KUKA KRL program: MyProgram_301().src

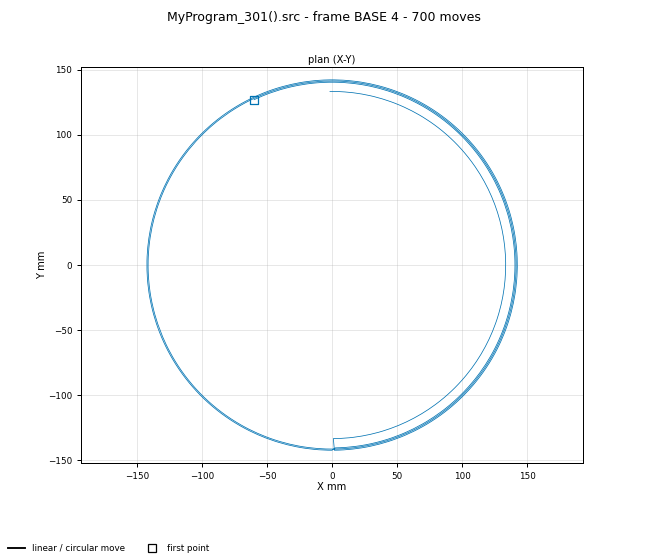
[picture p0: tool path of MyProgram_301().src in frame BASE 4, 700 of 700 moves have a stored position in this frame; points joined in program order, loops and branches not executed]
&ACCESS RVP
&REL 1
&PARAM TEMPLATE = C:\KRC\Roboter\Template\vorgabe
&PARAM EDITMASK = *
DEF MyProgram_301()
; ---- Setting reference (Base) ----
$BASE = BASE_DATA[4]

; --------------------------
; ---- Setting tool (TCP) ----
$TOOL = TOOL_DATA[3]
; --------------------------

$VEL.CP = VEL_APROX_PRINT
Startdeposition()
$VEL.CP = VEL_PRINT
LIN {X -59.9735,Y 127.061,Z 179,A 116.0898,B 5.4554,C 0.1242,E1 5.3915,E2 336.7382} C_DIS
LIN {X -56.1252,Y 128.8061,Z 179,A 114.464,B 5.4555,C 0.1213,E1 5.3956,E2 338.3506} C_DIS
LIN {X -53.7066,Y 129.8335,Z 179,A 112.9627,B 5.4555,C 0.1248,E1 5.3997,E2 339.9046} C_DIS
LIN {X -49.9072,Y 131.3417,Z 179,A 111.7575,B 5.4556,C 0.1181,E1 5.4027,E2 341.0513} C_DIS
LIN {X -46.6578,Y 132.5309,Z 179,A 110.2415,B 5.4556,C 0.1179,E1 5.4067,E2 342.5794} C_DIS
LIN {X -43.1664,Y 133.7078,Z 179,A 108.7239,B 5.4556,C 0.1168,E1 5.4107,E2 344.0979} C_DIS
LIN {X -39.9341,Y 134.7087,Z 179,A 107.5102,B 5.4557,C 0.1139,E1 5.4139,E2 345.2899} C_DIS
LIN {X -35.7865,Y 135.8693,Z 179,A 105.3832,B 5.4557,C 0.1168,E1 5.4197,E2 347.4621} C_DIS
LIN {X -31.4273,Y 136.9427,Z 179,A 103.8007,B 5.4557,C 0.1128,E1 5.4239,E2 349.0125} C_DIS
LIN {X -26.0499,Y 138.067,Z 179,A 101.4297,B 5.4557,C 0.1131,E1 5.4305,E2 351.3986} C_DIS
LIN {X -19.5272,Y 139.1395,Z 179,A 98.6974,B 5.4557,C 0.1125,E1 5.438,E2 354.1341} C_DIS
LIN {X -15.9211,Y 139.5996,Z 179,A 97.2765,B 5.4557,C 0.1113,E1 5.4419,E2 355.5466} C_DIS
LIN {X -11.8962,Y 139.9983,Z 179,A 95.031,B 5.4557,C 0.1179,E1 5.4484,E2 357.8653} C_DIS
LIN {X -6.6461,Y 140.3461,Z 179,A 93.5271,B 5.4557,C 0.1101,E1 5.4524,E2 359.2884} C_DIS
LIN {X -2.4559,Y 140.4815,Z 179,A 91.8062,B 5.4557,C 0.1102,E1 5.4572,E2 361.01} C_DIS
LIN {X 1.5144,Y 140.4967,Z 179,A 90.0682,B 5.4557,C 0.1117,E1 5.4621,E2 362.7621} C_DIS
LIN {X 5.4184,Y 140.3983,Z 179,A 88.5802,B 5.4557,C 0.1107,E1 5.4662,E2 364.2363} C_DIS
LIN {X 9.2875,Y 140.197,Z 179,A 86.9515,B 5.4557,C 0.1116,E1 5.4707,E2 365.8706} C_DIS
LIN {X 13.1744,Y 139.884,Z 179,A 85.4937,B 5.4557,C 0.1104,E1 5.4748,E2 367.3112} C_DIS
LIN {X 16.3822,Y 139.5446,Z 179,A 84.0811,B 5.4557,C 0.1121,E1 5.4787,E2 368.7355} C_DIS
LIN {X 22.469,Y 138.696,Z 179,A 81.6529,B 5.4557,C 0.1122,E1 5.4854,E2 371.1532} C_DIS
LIN {X 25.5598,Y 138.1606,Z 179,A 80.3615,B 5.4557,C 0.1131,E1 5.4889,E2 372.4458} C_DIS
LIN {X 29.0062,Y 137.4774,Z 179,A 78.85,B 5.4557,C 0.1149,E1 5.4931,E2 373.9666} C_DIS
LIN {X 36.0406,Y 135.8015,Z 179,A 75.9709,B 5.4557,C 0.1162,E1 5.5009,E2 376.8363} C_DIS
LIN {X 39.1776,Y 134.9302,Z 179,A 74.6743,B 5.4557,C 0.1169,E1 5.5044,E2 378.1288} C_DIS
LIN {X 42.5413,Y 133.9075,Z 179,A 73.2661,B 5.4557,C 0.1178,E1 5.5081,E2 379.5334} C_DIS
LIN {X 46.6696,Y 132.5268,Z 179,A 71.4197,B 5.4556,C 0.1204,E1 5.513,E2 381.3885} C_DIS
LIN {X 50.862,Y 130.9732,Z 179,A 69.7391,B 5.4556,C 0.1204,E1 5.5174,E2 383.0509} C_DIS
LIN {X 53.3945,Y 129.9638,Z 179,A 68.5414,B 5.4556,C 0.1228,E1 5.5205,E2 384.2594} C_DIS
LIN {X 57.312,Y 128.2819,Z 179,A 66.859,B 5.4555,C 0.1241,E1 5.5248,E2 385.9344} C_DIS
LIN {X 60.3668,Y 126.8731,Z 179,A 65.3438,B 5.4554,C 0.1277,E1 5.5287,E2 387.4675} C_DIS
LIN {X 65.3482,Y 124.3805,Z 179,A 63.2344,B 5.4554,C 0.1285,E1 5.5338,E2 389.5565} C_DIS
LIN {X 69.2323,Y 122.2642,Z 179,A 61.367,B 5.4553,C 0.1319,E1 5.5384,E2 391.432} C_DIS
LIN {X 73.1963,Y 119.9327,Z 179,A 59.5251,B 5.4553,C 0.1343,E1 5.5428,E2 393.2696} C_DIS
LIN {X 77.189,Y 117.4024,Z 179,A 57.7001,B 5.4553,C 0.1359,E1 5.5471,E2 395.0817} C_DIS
LIN {X 79.755,Y 115.6749,Z 179,A 56.1319,B 5.455,C 0.1422,E1 5.5508,E2 396.6886} C_DIS
LIN {X 82.8776,Y 113.4589,Z 179,A 54.84,B 5.455,C 0.1411,E1 5.5536,E2 397.9467} C_DIS
LIN {X 86.6009,Y 110.6427,Z 179,A 53.0145,B 5.455,C 0.1433,E1 5.5576,E2 399.7626} C_DIS
LIN {X 89.4387,Y 108.3616,Z 179,A 51.5047,B 5.455,C 0.1464,E1 5.5609,E2 401.2758} C_DIS
LIN {X 93.026,Y 105.2977,Z 179,A 49.9215,B 5.455,C 0.1452,E1 5.5642,E2 402.8161} C_DIS
LIN {X 96.3391,Y 102.2751,Z 179,A 47.5816,B 5.4547,C 0.156,E1 5.5691,E2 405.221} C_DIS
LIN {X 99.0644,Y 99.6378,Z 179,A 46.3542,B 5.4547,C 0.1546,E1 5.5715,E2 406.4084} C_DIS
LIN {X 102.2103,Y 96.4081,Z 179,A 44.5458,B 5.4547,C 0.1579,E1 5.575,E2 408.2135} C_DIS
LIN {X 105.3889,Y 92.923,Z 179,A 42.6665,B 5.4545,C 0.1614,E1 5.5785,E2 410.0877} C_DIS
LIN {X 108.7726,Y 88.9378,Z 179,A 40.4479,B 5.4543,C 0.1673,E1 5.5824,E2 412.318} C_DIS
LIN {X 111.8854,Y 84.99,Z 179,A 38.5181,B 5.4543,C 0.1702,E1 5.5857,E2 414.2331} C_DIS
LIN {X 114.5403,Y 81.3767,Z 179,A 36.8119,B 5.4542,C 0.1726,E1 5.5885,E2 415.9244} C_DIS
LIN {X 116.9616,Y 77.8554,Z 179,A 35.0581,B 5.454,C 0.1769,E1 5.5912,E2 417.6803} C_DIS
LIN {X 119.4477,Y 73.9851,Z 179,A 33.1916,B 5.4539,C 0.1813,E1 5.594,E2 419.5463} C_DIS
LIN {X 123.0392,Y 67.8445,Z 179,A 30.388,B 5.4537,C 0.187,E1 5.5979,E2 422.3387} C_DIS
LIN {X 125.0407,Y 64.0769,Z 179,A 28.7804,B 5.4537,C 0.1894,E1 5.6,E2 423.9302} C_DIS
LIN {X 126.7841,Y 60.5532,Z 179,A 27.2752,B 5.4535,C 0.1921,E1 5.6018,E2 425.4235} C_DIS
LIN {X 128.1026,Y 57.7127,Z 179,A 25.9599,B 5.4534,C 0.1959,E1 5.6033,E2 426.7445} C_DIS
LIN {X 129.3593,Y 54.842,Z 179,A 24.752,B 5.4533,C 0.1982,E1 5.6047,E2 427.9441} C_DIS
LIN {X 131.4521,Y 49.6125,Z 179,A 22.4725,B 5.4531,C 0.204,E1 5.607,E2 430.2225} C_DIS
LIN {X 132.5214,Y 46.685,Z 179,A 21.1591,B 5.4529,C 0.2081,E1 5.6082,E2 431.5422} C_DIS
LIN {X 133.8417,Y 42.7474,Z 179,A 19.6275,B 5.4529,C 0.2102,E1 5.6095,E2 433.0539} C_DIS
LIN {X 134.7772,Y 39.7003,Z 179,A 18.3035,B 5.4527,C 0.2141,E1 5.6106,E2 434.3818} C_DIS
LIN {X 135.6851,Y 36.4773,Z 179,A 16.9623,B 5.4526,C 0.2175,E1 5.6116,E2 435.7207} C_DIS
LIN {X 136.9654,Y 31.328,Z 179,A 15.0592,B 5.4525,C 0.2195,E1 5.6129,E2 437.5915} C_DIS
LIN {X 137.5627,Y 28.5976,Z 179,A 13.7924,B 5.4523,C 0.2246,E1 5.6136,E2 438.8755} C_DIS
LIN {X 138.2642,Y 24.9809,Z 179,A 12.2857,B 5.4521,C 0.2289,E1 5.6144,E2 440.3837} C_DIS
LIN {X 138.8135,Y 21.7222,Z 179,A 10.1318,B 5.4514,C 0.245,E1 5.6154,E2 442.6421} C_DIS
LIN {X 139.6771,Y 15.2107,Z 179,A 8.3722,B 5.4517,C 0.2385,E1 5.6159,E2 444.2856} C_DIS
LIN {X 140.0458,Y 11.3331,Z 179,A 6.7108,B 5.4514,C 0.2441,E1 5.6163,E2 445.9576} C_DIS
LIN {X 140.3011,Y 7.5426,Z 179,A 5.2604,B 5.4514,C 0.247,E1 5.6165,E2 447.3964} C_DIS
LIN {X 140.456,Y 3.6373,Z 179,A 3.6834,B 5.4511,C 0.2513,E1 5.6167,E2 448.9724} C_DIS
LIN {X 140.5034,Y -0.4635,Z 179,A 2.0429,B 5.4509,C 0.2556,E1 5.6167,E2 450.61} C_DIS
LIN {X 140.4368,Y -4.3279,Z 179,A 0.5019,B 5.4507,C 0.2595,E1 5.6166,E2 452.1476} C_DIS
LIN {X 140.2489,Y -8.4451,Z 179,A -1.064,B 5.4506,C 0.2625,E1 5.6164,E2 453.6999} C_DIS
LIN {X 139.9762,Y -12.1572,Z 179,A -2.5142,B 5.4504,C 0.2658,E1 5.616,E2 455.1425} C_DIS
LIN {X 139.5744,Y -16.133,Z 179,A -4.1622,B 5.4502,C 0.2707,E1 5.6155,E2 456.7942} C_DIS
LIN {X 139.1835,Y -19.2196,Z 179,A -5.448,B 5.45,C 0.2746,E1 5.6151,E2 458.0834} C_DIS
LIN {X 138.6268,Y -22.8834,Z 179,A -6.915,B 5.4498,C 0.2782,E1 5.6144,E2 459.5458} C_DIS
LIN {X 137.1833,Y -30.3685,Z 179,A -10.6169,B 5.4489,C 0.296,E1 5.6123,E2 463.3273} C_DIS
LIN {X 135.7517,Y -36.2274,Z 179,A -12.5921,B 5.4489,C 0.2954,E1 5.6109,E2 465.2418} C_DIS
LIN {X 134.7367,Y -39.8384,Z 179,A -13.9222,B 5.4489,C 0.2965,E1 5.6099,E2 466.5472} C_DIS
LIN {X 133.4221,Y -44.0409,Z 179,A -15.4975,B 5.4488,C 0.298,E1 5.6086,E2 468.0953} C_DIS
LIN {X 132.3787,Y -47.0869,Z 179,A -16.8262,B 5.4486,C 0.3018,E1 5.6073,E2 469.4272} C_DIS
LIN {X 131.1053,Y -50.5221,Z 179,A -18.223,B 5.4484,C 0.3044,E1 5.606,E2 470.8125} C_DIS
LIN {X 129.8345,Y -53.7041,Z 179,A -19.6741,B 5.4482,C 0.3089,E1 5.6044,E2 472.272} C_DIS
LIN {X 128.4058,Y -57.035,Z 179,A -21.053,B 5.448,C 0.3113,E1 5.6029,E2 473.6392} C_DIS
LIN {X 126.9294,Y -60.249,Z 179,A -22.4718,B 5.4478,C 0.3147,E1 5.6012,E2 475.0561} C_DIS
LIN {X 125.3758,Y -63.4187,Z 179,A -23.8583,B 5.4477,C 0.3176,E1 5.5995,E2 476.4369} C_DIS
LIN {X 123.5537,Y -66.9039,Z 179,A -25.5318,B 5.4474,C 0.3228,E1 5.5973,E2 478.1211} C_DIS
LIN {X 121.2798,Y -70.9418,Z 179,A -27.2877,B 5.4472,C 0.3255,E1 5.5949,E2 479.8611} C_DIS
LIN {X 117.8636,Y -76.4829,Z 179,A -29.9034,B 5.4468,C 0.3315,E1 5.591,E2 482.474} C_DIS
LIN {X 113.5484,Y -82.7547,Z 179,A -33.0276,B 5.4464,C 0.3392,E1 5.586,E2 485.6037} C_DIS
LIN {X 109.5829,Y -87.9384,Z 179,A -35.5981,B 5.4461,C 0.3439,E1 5.5816,E2 488.1645} C_DIS
LIN {X 106.9374,Y -91.1366,Z 179,A -37.2627,B 5.4459,C 0.3473,E1 5.5786,E2 489.827} C_DIS
LIN {X 104.9464,Y -93.4232,Z 179,A -38.4441,B 5.4457,C 0.3492,E1 5.5764,E2 491.0023} C_DIS
LIN {X 100.8459,Y -97.8345,Z 179,A -40.8197,B 5.4455,C 0.3533,E1 5.5719,E2 493.3694} C_DIS
LIN {X 97.8304,Y -100.8498,Z 179,A -42.5591,B 5.4452,C 0.3569,E1 5.5684,E2 495.1103} C_DIS
LIN {X 94.6187,Y -103.8693,Z 179,A -44.3238,B 5.445,C 0.36,E1 5.5648,E2 496.8723} C_DIS
LIN {X 90.594,Y -107.3979,Z 179,A -46.5101,B 5.4448,C 0.3643,E1 5.5602,E2 499.0609} C_DIS
LIN {X 87.1907,Y -110.1789,Z 179,A -48.2227,B 5.4446,C 0.3665,E1 5.5565,E2 500.7645} C_DIS
LIN {X 83.8356,Y -112.7522,Z 179,A -49.9475,B 5.4444,C 0.3696,E1 5.5527,E2 502.4908} C_DIS
LIN {X 77.9866,Y -116.874,Z 179,A -52.8046,B 5.4441,C 0.3737,E1 5.5461,E2 505.3422} C_DIS
LIN {X 72.6793,Y -120.2463,Z 179,A -55.5121,B 5.4437,C 0.3799,E1 5.5396,E2 508.0707} C_DIS
LIN {X 69.8696,Y -121.9007,Z 179,A -56.8094,B 5.4436,C 0.3814,E1 5.5365,E2 509.3649} C_DIS
LIN {X 65.3965,Y -124.3551,Z 179,A -58.5675,B 5.4436,C 0.3799,E1 5.5323,E2 511.0816} C_DIS
LIN {X 62.8045,Y -125.6861,Z 179,A -59.8854,B 5.4434,C 0.3834,E1 5.5289,E2 512.4178} C_DIS
LIN {X 59.2382,Y -127.4041,Z 179,A -61.3852,B 5.4434,C 0.3839,E1 5.5252,E2 513.9035} C_DIS
LIN {X 56.4868,Y -128.6498,Z 179,A -62.7339,B 5.4432,C 0.3871,E1 5.5217,E2 515.2688} C_DIS
LIN {X 52.7311,Y -130.2321,Z 179,A -64.274,B 5.4432,C 0.3874,E1 5.5178,E2 516.7938} C_DIS
LIN {X 49.4106,Y -131.5277,Z 179,A -65.7168,B 5.4431,C 0.3889,E1 5.514,E2 518.2363} C_DIS
LIN {X 46.2712,Y -132.6649,Z 179,A -66.9721,B 5.4431,C 0.3889,E1 5.5107,E2 519.4783} C_DIS
LIN {X 43.0135,Y -133.7567,Z 179,A -68.3877,B 5.4429,C 0.3905,E1 5.507,E2 520.8969} C_DIS
LIN {X 38.5766,Y -135.1051,Z 179,A -70.4033,B 5.4427,C 0.3939,E1 5.5015,E2 522.9304} C_DIS
LIN {X 34.6216,Y -136.1701,Z 179,A -72.4941,B 5.4422,C 0.401,E1 5.4957,E2 525.0779} C_DIS
LIN {X 29.928,Y -137.2784,Z 179,A -73.9126,B 5.4426,C 0.3951,E1 5.4921,E2 526.425} C_DIS
LIN {X 26.1079,Y -138.0559,Z 179,A -75.5015,B 5.4426,C 0.3962,E1 5.4877,E2 528.0148} C_DIS
LIN {X 22.1736,Y -138.7435,Z 179,A -77.5834,B 5.442,C 0.4031,E1 5.4818,E2 530.1578} C_DIS
LIN {X 17.83,Y -139.3675,Z 179,A -78.9522,B 5.4424,C 0.3985,E1 5.4781,E2 531.4719} C_DIS
LIN {X 13.6739,Y -139.836,Z 179,A -80.5373,B 5.4424,C 0.3976,E1 5.4738,E2 533.0418} C_DIS
LIN {X 10.8007,Y -140.0882,Z 179,A -81.8644,B 5.4423,C 0.4,E1 5.47,E2 534.3897} C_DIS
LIN {X 6.6782,Y -140.3445,Z 179,A -83.5282,B 5.4423,C 0.4002,E1 5.4654,E2 536.0516} C_DIS
LIN {X 2.5643,Y -140.4797,Z 179,A -85.0032,B 5.4424,C 0.3979,E1 5.4613,E2 537.5002} C_DIS
LIN {X 2.5643,Y -140.4797,Z 179,A -85.0032,B 5.4424,C 0.3979,E1 5.4613,E2 537.5002} C_DIS
Enddeposition()
LIN {X 0.9995,Y -141.4027,Z 179,A -85.5688,B 5.4422,C 0.4002,E1 5.4597,E2 538.089} C_DIS
Startdeposition()
$VEL.CP = VEL_PRINT
LIN {X 4.3079,Y -141.3411,Z 179,A -83.7777,B 5.4426,C 0.3941,E1 5.4648,E2 536.2364} C_DIS
LIN {X 8.0416,Y -141.1788,Z 179,A -82.3225,B 5.4426,C 0.3945,E1 5.4689,E2 534.7885} C_DIS
LIN {X 10.4771,Y -141.0176,Z 179,A -81.2424,B 5.4427,C 0.393,E1 5.4719,E2 533.6954} C_DIS
LIN {X 13.695,Y -140.7415,Z 179,A -79.9223,B 5.4427,C 0.3923,E1 5.4756,E2 532.3731} C_DIS
LIN {X 18.1055,Y -140.2424,Z 179,A -78.054,B 5.4429,C 0.3905,E1 5.4808,E2 530.4943} C_DIS
LIN {X 21.9939,Y -139.6855,Z 179,A -76.6375,B 5.4428,C 0.392,E1 5.4847,E2 529.1007} C_DIS
LIN {X 25.7892,Y -139.0366,Z 179,A -75.0635,B 5.4428,C 0.3909,E1 5.489,E2 527.524} C_DIS
LIN {X 28.3252,Y -138.54,Z 179,A -73.9262,B 5.443,C 0.3889,E1 5.4921,E2 526.3737} C_DIS
LIN {X 34.9333,Y -137.023,Z 179,A -71.2683,B 5.443,C 0.388,E1 5.4994,E2 523.7262} C_DIS
LIN {X 38.5958,Y -136.0377,Z 179,A -69.4507,B 5.4434,C 0.3828,E1 5.5043,E2 521.8694} C_DIS
LIN {X 41.7903,Y -135.0902,Z 179,A -68.4169,B 5.4432,C 0.3859,E1 5.507,E2 520.8777} C_DIS
LIN {X 45.0381,Y -134.0422,Z 179,A -66.9833,B 5.4434,C 0.3838,E1 5.5108,E2 519.4363} C_DIS
LIN {X 48.6768,Y -132.7657,Z 179,A -65.4951,B 5.4434,C 0.3831,E1 5.5147,E2 517.9571} C_DIS
LIN {X 51.5748,Y -131.6653,Z 179,A -64.2322,B 5.4435,C 0.3816,E1 5.518,E2 516.6923} C_DIS
LIN {X 55.4697,Y -130.0737,Z 179,A -62.6111,B 5.4435,C 0.3807,E1 5.5221,E2 515.0813} C_DIS
LIN {X 58.2837,Y -128.8368,Z 179,A -61.3322,B 5.4437,C 0.3787,E1 5.5254,E2 513.797} C_DIS
LIN {X 61.5935,Y -127.2882,Z 179,A -59.8657,B 5.4439,C 0.3769,E1 5.5291,E2 512.3313} C_DIS
LIN {X 64.4708,Y -125.8538,Z 179,A -58.5722,B 5.4439,C 0.3752,E1 5.5323,E2 511.038} C_DIS
LIN {X 67.6591,Y -124.1708,Z 179,A -56.614,B 5.4446,C 0.3659,E1 5.5373,E2 509.011} C_DIS
LIN {X 71.7411,Y -121.8579,Z 179,A -55.1964,B 5.4443,C 0.37,E1 5.5406,E2 507.6577} C_DIS
LIN {X 75.4899,Y -119.5717,Z 179,A -53.4446,B 5.4445,C 0.3676,E1 5.5447,E2 505.9083} C_DIS
LIN {X 79.2527,Y -117.1116,Z 179,A -51.5254,B 5.4448,C 0.3631,E1 5.5492,E2 503.9742} C_DIS
LIN {X 82.4628,Y -114.8741,Z 179,A -50.2247,B 5.4447,C 0.3646,E1 5.5521,E2 502.7109} C_DIS
LIN {X 85.389,Y -112.716,Z 179,A -48.6509,B 5.445,C 0.3604,E1 5.5557,E2 501.1222} C_DIS
LIN {X 88.4591,Y -110.3235,Z 179,A -47.0465,B 5.4452,C 0.3571,E1 5.5592,E2 499.5128} C_DIS
LIN {X 91.7741,Y -107.5811,Z 179,A -45.3391,B 5.4454,C 0.3543,E1 5.5628,E2 497.8088} C_DIS
LIN {X 95.2955,Y -104.475,Z 179,A -43.5116,B 5.4455,C 0.3517,E1 5.5666,E2 495.9898} C_DIS
LIN {X 98.3118,Y -101.6411,Z 179,A -41.8441,B 5.4457,C 0.3484,E1 5.57,E2 494.3221} C_DIS
LIN {X 101.5,Y -98.4575,Z 179,A -39.9945,B 5.446,C 0.3442,E1 5.5736,E2 492.4676} C_DIS
LIN {X 104.7884,Y -94.95,Z 179,A -38.1227,B 5.4462,C 0.3411,E1 5.5771,E2 490.6045} C_DIS
LIN {X 107.6795,Y -91.6583,Z 179,A -36.4504,B 5.4464,C 0.3388,E1 5.5802,E2 488.9445} C_DIS
LIN {X 110.2359,Y -88.5677,Z 179,A -34.7304,B 5.4467,C 0.3336,E1 5.5832,E2 487.2102} C_DIS
LIN {X 114.336,Y -83.2074,Z 179,A -32.4216,B 5.4467,C 0.3338,E1 5.587,E2 484.9564} C_DIS
LIN {X 117.0989,Y -79.2715,Z 179,A -30.2178,B 5.4472,C 0.3252,E1 5.5906,E2 482.7165} C_DIS
LIN {X 119.5465,Y -75.5298,Z 179,A -28.2286,B 5.4476,C 0.318,E1 5.5936,E2 480.7017} C_DIS
LIN {X 121.3857,Y -72.5372,Z 179,A -27.19,B 5.4475,C 0.3204,E1 5.595,E2 479.7137} C_DIS
LIN {X 123.3717,Y -69.1057,Z 179,A -25.5315,B 5.4477,C 0.3156,E1 5.5973,E2 478.0467} C_DIS
LIN {X 125.4173,Y -65.3168,Z 179,A -23.8624,B 5.4479,C 0.3123,E1 5.5995,E2 476.3861} C_DIS
LIN {X 126.9466,Y -62.2912,Z 179,A -22.5008,B 5.4481,C 0.3089,E1 5.6012,E2 475.025} C_DIS
LIN {X 128.5114,Y -58.9959,Z 179,A -21.0728,B 5.4483,C 0.3058,E1 5.6029,E2 473.6024} C_DIS
LIN {X 129.9129,Y -55.8417,Z 179,A -19.6603,B 5.4485,C 0.3019,E1 5.6045,E2 472.1868} C_DIS
LIN {X 131.3582,Y -52.3535,Z 179,A -18.2356,B 5.4486,C 0.2995,E1 5.606,E2 470.7748} C_DIS
LIN {X 132.4579,Y -49.5025,Z 179,A -16.9874,B 5.4488,C 0.296,E1 5.6072,E2 469.5241} C_DIS
LIN {X 133.8629,Y -45.5732,Z 179,A -15.381,B 5.449,C 0.2927,E1 5.6087,E2 467.9277} C_DIS
LIN {X 134.7945,Y -42.7332,Z 179,A -13.5688,B 5.4497,C 0.2799,E1 5.6103,E2 466.0335} C_DIS
LIN {X 136.3125,Y -37.6132,Z 179,A -12.1345,B 5.4494,C 0.2855,E1 5.6113,E2 464.6954} C_DIS
LIN {X 137.1844,Y -34.2974,Z 179,A -10.7171,B 5.4496,C 0.2812,E1 5.6123,E2 463.2731} C_DIS
LIN {X 138.048,Y -30.6439,Z 179,A -9.2203,B 5.4498,C 0.2773,E1 5.6132,E2 461.7783} C_DIS
LIN {X 138.9256,Y -26.3697,Z 179,A -7.5013,B 5.45,C 0.2731,E1 5.6141,E2 460.0642} C_DIS
LIN {X 139.5935,Y -22.5785,Z 179,A -5.8441,B 5.4503,C 0.2672,E1 5.6149,E2 458.3928} C_DIS
LIN {X 140.2021,Y -18.4129,Z 179,A -4.2597,B 5.4505,C 0.2643,E1 5.6155,E2 456.8231} C_DIS
LIN {X 140.6466,Y -14.6442,Z 179,A -2.862,B 5.4505,C 0.2621,E1 5.6159,E2 455.4428} C_DIS
LIN {X 140.9084,Y -11.8539,Z 179,A -1.7325,B 5.4507,C 0.259,E1 5.6162,E2 454.3132} C_DIS
LIN {X 141.1762,Y -8.0844,Z 179,A -0.2635,B 5.4509,C 0.2556,E1 5.6164,E2 452.8513} C_DIS
LIN {X 141.3108,Y -5.2017,Z 179,A 0.8759,B 5.451,C 0.2527,E1 5.6166,E2 451.7149} C_DIS
LIN {X 141.3956,Y -1.8135,Z 179,A 2.3343,B 5.4512,C 0.2475,E1 5.6166,E2 450.2441} C_DIS
LIN {X 141.3891,Y 2.2053,Z 179,A 3.8559,B 5.4514,C 0.2445,E1 5.6166,E2 448.7354} C_DIS
LIN {X 141.2762,Y 6.0877,Z 179,A 5.3231,B 5.4515,C 0.2417,E1 5.6165,E2 447.2812} C_DIS
LIN {X 141.092,Y 9.4502,Z 179,A 6.8304,B 5.4518,C 0.2356,E1 5.6162,E2 445.754} C_DIS
LIN {X 140.7421,Y 13.6884,Z 179,A 8.4336,B 5.4519,C 0.2326,E1 5.6158,E2 444.1654} C_DIS
LIN {X 140.0507,Y 19.5367,Z 179,A 10.5523,B 5.452,C 0.23,E1 5.6151,E2 442.0804} C_DIS
LIN {X 139.6935,Y 21.9426,Z 179,A 11.7579,B 5.4523,C 0.2238,E1 5.6146,E2 440.845} C_DIS
LIN {X 139.0271,Y 25.8385,Z 179,A 13.1623,B 5.4523,C 0.2224,E1 5.6139,E2 439.4656} C_DIS
LIN {X 138.0468,Y 30.6493,Z 179,A 15.1393,B 5.4525,C 0.2171,E1 5.6127,E2 437.489} C_DIS
LIN {X 137.4441,Y 33.238,Z 179,A 16.1352,B 5.4526,C 0.2153,E1 5.6121,E2 436.503} C_DIS
LIN {X 136.5242,Y 36.8366,Z 179,A 17.791,B 5.4529,C 0.2089,E1 5.6109,E2 434.8264} C_DIS
LIN {X 135.1491,Y 41.5978,Z 179,A 19.6956,B 5.453,C 0.205,E1 5.6094,E2 432.9342} C_DIS
LIN {X 133.9089,Y 45.4383,Z 179,A 21.2219,B 5.4531,C 0.2023,E1 5.6081,E2 431.4214} C_DIS
LIN {X 132.8684,Y 48.392,Z 179,A 22.4659,B 5.4532,C 0.1992,E1 5.6069,E2 430.1798} C_DIS
LIN {X 131.3335,Y 52.4149,Z 179,A 24.0987,B 5.4533,C 0.1963,E1 5.6053,E2 428.5608} C_DIS
LIN {X 129.9658,Y 55.7193,Z 179,A 25.7295,B 5.4536,C 0.1897,E1 5.6035,E2 426.9053} C_DIS
LIN {X 128.1395,Y 59.8002,Z 179,A 27.374,B 5.4536,C 0.1876,E1 5.6016,E2 425.2818} C_DIS
LIN {X 126.6554,Y 62.8816,Z 179,A 28.709,B 5.4537,C 0.1848,E1 5.5999,E2 423.9528} C_DIS
LIN {X 124.9198,Y 66.2642,Z 179,A 30.2338,B 5.4538,C 0.1812,E1 5.598,E2 422.4294} C_DIS
LIN {X 122.5344,Y 70.58,Z 179,A 31.9634,B 5.4538,C 0.1803,E1 5.5957,E2 420.734} C_DIS
LIN {X 121.1409,Y 72.9456,Z 179,A 33.3015,B 5.4541,C 0.1742,E1 5.5937,E2 419.366} C_DIS
LIN {X 118.9743,Y 76.4283,Z 179,A 34.8972,B 5.4541,C 0.1712,E1 5.5913,E2 417.7782} C_DIS
LIN {X 116.8132,Y 79.6928,Z 179,A 36.5251,B 5.4543,C 0.1668,E1 5.5888,E2 416.1443} C_DIS
LIN {X 114.1533,Y 83.4581,Z 179,A 38.3746,B 5.4544,C 0.1627,E1 5.5858,E2 414.2966} C_DIS
LIN {X 111.3389,Y 87.1769,Z 179,A 41.0152,B 5.4549,C 0.1473,E1 5.5811,E2 411.5569} C_DIS
LIN {X 106.9212,Y 92.5423,Z 179,A 42.6786,B 5.4546,C 0.1582,E1 5.5783,E2 410.0434} C_DIS
LIN {X 104.2774,Y 95.5113,Z 179,A 44.5475,B 5.4548,C 0.151,E1 5.5748,E2 408.1407} C_DIS
LIN {X 101.2022,Y 98.7642,Z 179,A 46.3398,B 5.4548,C 0.1476,E1 5.5713,E2 406.3508} C_DIS
LIN {X 92.8002,Y 106.6972,Z 179,A 50.5701,B 5.4549,C 0.145,E1 5.5628,E2 402.1783} C_DIS
LIN {X 90.2409,Y 108.8701,Z 179,A 52.0081,B 5.455,C 0.1414,E1 5.5597,E2 400.7302} C_DIS
LIN {X 87.7377,Y 110.8981,Z 179,A 53.57,B 5.4552,C 0.1354,E1 5.5562,E2 399.1351} C_DIS
LIN {X 84.0274,Y 113.735,Z 179,A 55.4478,B 5.4552,C 0.1323,E1 5.552,E2 397.259} C_DIS
LIN {X 80.1939,Y 116.4693,Z 179,A 57.2469,B 5.4552,C 0.1307,E1 5.5479,E2 395.4738} C_DIS
LIN {X 76.7917,Y 118.7402,Z 179,A 58.8582,B 5.4553,C 0.1287,E1 5.5442,E2 393.8683} C_DIS
LIN {X 73.4381,Y 120.8431,Z 179,A 60.4892,B 5.4553,C 0.1259,E1 5.5403,E2 392.2339} C_DIS
LIN {X 69.5643,Y 123.1139,Z 179,A 62.3138,B 5.4555,C 0.1232,E1 5.5359,E2 390.4085} C_DIS
LIN {X 63.6906,Y 126.251,Z 179,A 64.8495,B 5.4555,C 0.1218,E1 5.5297,E2 387.8938} C_DIS
LIN {X 60.3586,Y 127.8782,Z 179,A 66.3343,B 5.4555,C 0.1201,E1 5.5259,E2 386.4114} C_DIS
LIN {X 57.216,Y 129.3144,Z 179,A 67.8739,B 5.4556,C 0.1166,E1 5.522,E2 384.8541} C_DIS
LIN {X 53.6713,Y 130.8269,Z 179,A 69.2707,B 5.4556,C 0.117,E1 5.5184,E2 383.4787} C_DIS
LIN {X 50.8579,Y 131.944,Z 179,A 70.5007,B 5.4556,C 0.1157,E1 5.5152,E2 382.2483} C_DIS
LIN {X 47.5256,Y 133.1807,Z 179,A 72.1401,B 5.4557,C 0.1116,E1 5.5109,E2 380.5835} C_DIS
LIN {X 43.1876,Y 134.6494,Z 179,A 73.8845,B 5.4557,C 0.1113,E1 5.5063,E2 378.8538} C_DIS
LIN {X 38.9181,Y 135.9474,Z 179,A 75.5456,B 5.4557,C 0.1118,E1 5.5019,E2 377.2121} C_DIS
LIN {X 34.6025,Y 137.107,Z 179,A 77.4304,B 5.4557,C 0.1094,E1 5.4967,E2 375.318} C_DIS
LIN {X 30.5262,Y 138.0734,Z 179,A 78.9833,B 5.4557,C 0.1101,E1 5.4926,E2 373.7842} C_DIS
LIN {X 28.1021,Y 138.5854,Z 179,A 80.1016,B 5.4557,C 0.1081,E1 5.4895,E2 372.6514} C_DIS
LIN {X 24.3134,Y 139.3014,Z 179,A 81.5785,B 5.4557,C 0.1083,E1 5.4854,E2 371.186} C_DIS
LIN {X 19.7106,Y 140.0258,Z 179,A 83.4815,B 5.4557,C 0.1072,E1 5.4802,E2 369.2816} C_DIS
LIN {X 16.3303,Y 140.4606,Z 179,A 84.7817,B 5.4557,C 0.1077,E1 5.4766,E2 367.9923} C_DIS
LIN {X 13.2086,Y 140.7882,Z 179,A 86.2109,B 5.4558,C 0.1053,E1 5.4726,E2 366.5434} C_DIS
LIN {X 8.9197,Y 141.1247,Z 179,A 87.9047,B 5.4558,C 0.1055,E1 5.4679,E2 364.8566} C_DIS
LIN {X 5.0338,Y 141.3174,Z 179,A 89.5584,B 5.4558,C 0.1043,E1 5.4632,E2 363.1937} C_DIS
LIN {X 0.5177,Y 141.4055,Z 179,A 91.3077,B 5.4558,C 0.1052,E1 5.4584,E2 361.4555} C_DIS
LIN {X -3.1022,Y 141.3742,Z 179,A 92.6987,B 5.4558,C 0.1061,E1 5.4545,E2 360.0749} C_DIS
LIN {X -6.3182,Y 141.2671,Z 179,A 94.2803,B 5.4558,C 0.1029,E1 5.45,E2 358.4584} C_DIS
LIN {X -10.6336,Y 141.0061,Z 179,A 95.7763,B 5.4558,C 0.1062,E1 5.4459,E2 356.996} C_DIS
LIN {X -14.818,Y 140.6279,Z 179,A 97.4476,B 5.4558,C 0.107,E1 5.4413,E2 355.3295} C_DIS
LIN {X -17.7046,Y 140.2949,Z 179,A 98.7868,B 5.4558,C 0.1054,E1 5.4375,E2 353.9702} C_DIS
LIN {X -22.2365,Y 139.6475,Z 179,A 101.0043,B 5.4558,C 0.1019,E1 5.4313,E2 351.7073} C_DIS
LIN {X -26.4875,Y 138.903,Z 179,A 102.3477,B 5.4558,C 0.1075,E1 5.4277,E2 350.4168} C_DIS
LIN {X -30.1852,Y 138.147,Z 179,A 103.8422,B 5.4558,C 0.1087,E1 5.4237,E2 348.9277} C_DIS
LIN {X -34.2779,Y 137.1893,Z 179,A 106.1026,B 5.4558,C 0.1034,E1 5.4174,E2 346.5968} C_DIS
LIN {X -39.0294,Y 135.9148,Z 179,A 107.4949,B 5.4558,C 0.1118,E1 5.4138,E2 345.283} C_DIS
LIN {X -42.3801,Y 134.9073,Z 179,A 108.9044,B 5.4557,C 0.113,E1 5.4101,E2 343.8754} C_DIS
LIN {X -45.1784,Y 133.9954,Z 179,A 110.173,B 5.4557,C 0.1132,E1 5.4067,E2 342.5978} C_DIS
LIN {X -49.121,Y 132.6008,Z 179,A 112.0412,B 5.4557,C 0.1128,E1 5.4017,E2 340.7086} C_DIS
LIN {X -52.9605,Y 131.1136,Z 179,A 113.6582,B 5.4557,C 0.1151,E1 5.3975,E2 339.0993} C_DIS
LIN {X -56.4558,Y 129.6474,Z 179,A 115.1341,B 5.4556,C 0.1174,E1 5.3938,E2 337.6321} C_DIS
LIN {X -59.8038,Y 128.1379,Z 179,A 116.6459,B 5.4556,C 0.1189,E1 5.3899,E2 336.1184} C_DIS
LIN {X -63.3872,Y 126.4055,Z 179,A 118.255,B 5.4556,C 0.1209,E1 5.3859,E2 334.5109} C_DIS
LIN {X -67.0537,Y 124.4988,Z 179,A 120.0426,B 5.4555,C 0.1219,E1 5.3814,E2 332.7101} C_DIS
LIN {X -71.0188,Y 122.2804,Z 179,A 121.9262,B 5.4555,C 0.124,E1 5.3769,E2 330.8224} C_DIS
LIN {X -75.0441,Y 119.8527,Z 179,A 123.8601,B 5.4554,C 0.1265,E1 5.3723,E2 328.8862} C_DIS
LIN {X -78.9175,Y 117.3385,Z 179,A 125.7741,B 5.4554,C 0.1289,E1 5.3678,E2 326.9682} C_DIS
LIN {X -85.6625,Y 112.5084,Z 179,A 128.8659,B 5.4551,C 0.1373,E1 5.3609,E2 323.9138} C_DIS
LIN {X -87.9222,Y 110.7513,Z 179,A 130.2927,B 5.4551,C 0.1365,E1 5.3577,E2 322.4538} C_DIS
LIN {X -91.1943,Y 108.0735,Z 179,A 132.4097,B 5.4551,C 0.1355,E1 5.353,E2 320.2863} C_DIS
LIN {X -94.2464,Y 105.4217,Z 179,A 133.904,B 5.4551,C 0.1401,E1 5.35,E2 318.8119} C_DIS
LIN {X -98.227,Y 101.7232,Z 179,A 136.0031,B 5.4549,C 0.1454,E1 5.3457,E2 316.7278} C_DIS
LIN {X -101.5761,Y 98.379,Z 179,A 138.2849,B 5.4549,C 0.1456,E1 5.3412,E2 314.4008} C_DIS
LIN {X -104.4166,Y 95.359,Z 179,A 139.7378,B 5.4548,C 0.1514,E1 5.3385,E2 312.9786} C_DIS
LIN {X -110.3474,Y 88.4294,Z 179,A 144.2085,B 5.4548,C 0.1518,E1 5.3304,E2 308.4106} C_DIS
LIN {X -114.2965,Y 83.2619,Z 179,A 145.8305,B 5.4543,C 0.1677,E1 5.3279,E2 306.9223} C_DIS
LIN {X -117.2668,Y 79.0235,Z 179,A 148.1978,B 5.4543,C 0.17,E1 5.3241,E2 304.5221} C_DIS
LIN {X -119.6034,Y 75.4398,Z 179,A 150.051,B 5.4541,C 0.173,E1 5.3213,E2 302.6549} C_DIS
LIN {X -122.0106,Y 71.4813,Z 179,A 151.9552,B 5.454,C 0.1774,E1 5.3185,E2 300.7489} C_DIS
LIN {X -124.3232,Y 67.3797,Z 179,A 154.1234,B 5.4539,C 0.1796,E1 5.3156,E2 298.5487} C_DIS
LIN {X -125.8307,Y 64.5163,Z 179,A 155.4705,B 5.4538,C 0.1826,E1 5.3139,E2 297.198} C_DIS
LIN {X -127.3722,Y 61.4177,Z 179,A 156.4633,B 5.4535,C 0.1901,E1 5.3127,E2 296.2594} C_DIS
LIN {X -129.2797,Y 57.2935,Z 179,A 158.5152,B 5.4535,C 0.1929,E1 5.3103,E2 294.1819} C_DIS
LIN {X -131.5415,Y 51.8933,Z 179,A 160.8546,B 5.4532,C 0.1995,E1 5.3078,E2 291.849} C_DIS
LIN {X -132.5521,Y 49.2509,Z 179,A 162.1209,B 5.4532,C 0.2014,E1 5.3066,E2 290.568} C_DIS
LIN {X -133.6876,Y 46.0789,Z 179,A 163.4986,B 5.453,C 0.2049,E1 5.3053,E2 289.1899} C_DIS
LIN {X -134.7082,Y 43.0035,Z 179,A 164.8781,B 5.4529,C 0.2079,E1 5.3041,E2 287.8028} C_DIS
LIN {X -135.9946,Y 38.7499,Z 179,A 166.6216,B 5.4527,C 0.2133,E1 5.3027,E2 286.0684} C_DIS
LIN {X -136.7897,Y 35.8407,Z 179,A 167.9215,B 5.4526,C 0.216,E1 5.3018,E2 284.7594} C_DIS
LIN {X -137.5055,Y 32.9831,Z 179,A 169.1618,B 5.4525,C 0.2189,E1 5.301,E2 283.5141} C_DIS
LIN {X -138.295,Y 29.4999,Z 179,A 171.3606,B 5.4525,C 0.2159,E1 5.2996,E2 281.2181} C_DIS
LIN {X -139.3643,Y 23.9522,Z 179,A 172.936,B 5.4521,C 0.229,E1 5.2989,E2 279.7382} C_DIS
LIN {X -139.7776,Y 21.3995,Z 179,A 174.1256,B 5.452,C 0.2306,E1 5.2984,E2 278.531} C_DIS
LIN {X -140.3853,Y 16.9614,Z 179,A 176.3124,B 5.452,C 0.2323,E1 5.2976,E2 276.297} C_DIS
LIN {X -140.7863,Y 13.2281,Z 179,A 177.5696,B 5.4516,C 0.2391,E1 5.2973,E2 275.0756} C_DIS
LIN {X -141.0724,Y 9.7259,Z 179,A 178.9252,B 5.4514,C 0.2437,E1 5.297,E2 273.73} C_DIS
LIN {X -141.2632,Y 6.3954,Z 179,A -179.6842,B 5.4513,C 0.2472,E1 5.2968,E2 272.3355} C_DIS
LIN {X -141.3607,Y 3.6021,Z 179,A -178.4224,B 5.4512,C 0.2493,E1 5.2967,E2 271.0576} C_DIS
LIN {X -141.3989,Y -1.5802,Z 179,A -176.0952,B 5.451,C 0.2531,E1 5.2967,E2 268.7022} C_DIS
LIN {X -141.2996,Y -5.4889,Z 179,A -174.635,B 5.4507,C 0.2588,E1 5.2968,E2 267.2595} C_DIS
LIN {X -141.0719,Y -9.7334,Z 179,A -172.7693,B 5.4506,C 0.2623,E1 5.2972,E2 265.3762} C_DIS
LIN {X -140.4728,Y -16.2277,Z 179,A -170.1651,B 5.4502,C 0.2702,E1 5.2979,E2 262.779} C_DIS
LIN {X -139.8416,Y -20.9861,Z 179,A -168.096,B 5.45,C 0.2745,E1 5.2987,E2 260.6949} C_DIS
LIN {X -139.3131,Y -24.248,Z 179,A -166.5884,B 5.4498,C 0.2766,E1 5.2994,E2 259.166} C_DIS
LIN {X -138.436,Y -28.8366,Z 179,A -164.9004,B 5.4495,C 0.2838,E1 5.3003,E2 257.5062} C_DIS
LIN {X -137.7649,Y -31.8844,Z 179,A -163.6107,B 5.4493,C 0.2871,E1 5.3011,E2 256.214} C_DIS
LIN {X -137.0373,Y -34.8771,Z 179,A -162.3238,B 5.4491,C 0.2901,E1 5.302,E2 254.9228} C_DIS
LIN {X -136.1721,Y -38.1152,Z 179,A -160.8821,B 5.449,C 0.293,E1 5.3031,E2 253.4708} C_DIS
LIN {X -134.9073,Y -42.3801,Z 179,A -159.143,B 5.4487,C 0.2985,E1 5.3045,E2 251.7413} C_DIS
LIN {X -133.9887,Y -45.1988,Z 179,A -157.8305,B 5.4486,C 0.3007,E1 5.3056,E2 250.4148} C_DIS
LIN {X -131.0661,Y -53.0783,Z 179,A -154.7493,B 5.4479,C 0.3128,E1 5.3086,E2 247.3784} C_DIS
LIN {X -130.2875,Y -54.9635,Z 179,A -153.4872,B 5.448,C 0.3108,E1 5.31,E2 246.0592} C_DIS
LIN {X -128.4471,Y -59.135,Z 179,A -151.8434,B 5.4476,C 0.3175,E1 5.3119,E2 244.4434} C_DIS
LIN {X -127.4658,Y -61.2217,Z 179,A -150.6354,B 5.4476,C 0.3172,E1 5.3134,E2 243.1996} C_DIS
LIN {X -125.6976,Y -64.7778,Z 179,A -148.9922,B 5.4474,C 0.3209,E1 5.3154,E2 241.5527} C_DIS
LIN {X -122.7235,Y -70.2504,Z 179,A -146.456,B 5.4471,C 0.327,E1 5.3189,E2 239.0161} C_DIS
LIN {X -120.7719,Y -73.5559,Z 179,A -144.7303,B 5.4469,C 0.329,E1 5.3214,E2 237.2683} C_DIS
LIN {X -118.3289,Y -77.4245,Z 179,A -142.8303,B 5.4467,C 0.3329,E1 5.3243,E2 235.363} C_DIS
LIN {X -115.767,Y -81.2051,Z 179,A -141.0106,B 5.4464,C 0.3374,E1 5.3271,E2 233.548} C_DIS
LIN {X -113.1811,Y -84.7722,Z 179,A -139.1586,B 5.4462,C 0.3407,E1 5.3302,E2 231.6877} C_DIS
LIN {X -110.6783,Y -88.0138,Z 179,A -137.4354,B 5.446,C 0.3437,E1 5.3332,E2 229.9565} C_DIS
LIN {X -107.754,Y -91.5707,Z 179,A -135.5278,B 5.4458,C 0.3472,E1 5.3366,E2 228.0438} C_DIS
LIN {X -104.8282,Y -94.9062,Z 179,A -133.6848,B 5.4456,C 0.3504,E1 5.3401,E2 226.1953} C_DIS
LIN {X -101.6507,Y -98.3019,Z 179,A -131.767,B 5.4454,C 0.3539,E1 5.3438,E2 224.2734} C_DIS
LIN {X -98.272,Y -101.6796,Z 179,A -129.8116,B 5.4452,C 0.3574,E1 5.3477,E2 222.3158} C_DIS
LIN {X -94.9086,Y -104.8261,Z 179,A -127.9305,B 5.4449,C 0.3607,E1 5.3515,E2 220.433} C_DIS
LIN {X -91.6647,Y -107.6741,Z 179,A -126.156,B 5.4448,C 0.3635,E1 5.3553,E2 218.6554} C_DIS
LIN {X -88.4076,Y -110.3649,Z 179,A -124.3717,B 5.4446,C 0.3656,E1 5.3592,E2 216.8616} C_DIS
LIN {X -84.3361,Y -113.5058,Z 179,A -122.4295,B 5.4443,C 0.3706,E1 5.3635,E2 214.9386} C_DIS
LIN {X -81.2673,Y -115.7231,Z 179,A -120.7232,B 5.4443,C 0.3711,E1 5.3674,E2 213.2092} C_DIS
LIN {X -77.4426,Y -118.317,Z 179,A -118.8712,B 5.444,C 0.3741,E1 5.3717,E2 211.3601} C_DIS
LIN {X -73.7782,Y -120.6356,Z 179,A -117.0476,B 5.444,C 0.3758,E1 5.376,E2 209.5275} C_DIS
LIN {X -69.8871,Y -122.9307,Z 179,A -114.9801,B 5.444,C 0.3756,E1 5.3811,E2 207.428} C_DIS
LIN {X -66.9346,Y -124.5628,Z 179,A -113.973,B 5.4435,C 0.3814,E1 5.3835,E2 206.4695} C_DIS
LIN {X -63.8442,Y -126.1728,Z 179,A -112.448,B 5.4435,C 0.3818,E1 5.3873,E2 204.929} C_DIS
LIN {X -60.3054,Y -127.9036,Z 179,A -110.8447,B 5.4434,C 0.3835,E1 5.3913,E2 203.3247} C_DIS
LIN {X -57.4714,Y -129.2002,Z 179,A -109.568,B 5.4434,C 0.3847,E1 5.3946,E2 202.0458} C_DIS
LIN {X -53.9333,Y -130.7178,Z 179,A -108.0188,B 5.4432,C 0.3863,E1 5.3986,E2 200.498} C_DIS
LIN {X -51.0028,Y -131.8876,Z 179,A -106.365,B 5.4434,C 0.3831,E1 5.403,E2 198.7931} C_DIS
LIN {X -47.5098,Y -133.1864,Z 179,A -104.878,B 5.4434,C 0.3846,E1 5.4069,E2 197.309} C_DIS
LIN {X -44.2066,Y -134.3191,Z 179,A -103.7565,B 5.443,C 0.3892,E1 5.4098,E2 196.227} C_DIS
LIN {X -39.8549,Y -135.6731,Z 179,A -101.7584,B 5.443,C 0.3887,E1 5.4152,E2 194.208} C_DIS
LIN {X -35.7977,Y -136.8012,Z 179,A -100.2132,B 5.4428,C 0.3917,E1 5.4193,E2 192.6842} C_DIS
LIN {X -32.749,Y -137.5619,Z 179,A -98.9596,B 5.4428,C 0.3927,E1 5.4227,E2 191.4328} C_DIS
LIN {X -29.1283,Y -138.3752,Z 179,A -97.4128,B 5.4428,C 0.3929,E1 5.4269,E2 189.8799} C_DIS
LIN {X -26.1918,Y -138.9596,Z 179,A -96.1374,B 5.4428,C 0.3926,E1 5.4305,E2 188.5956} C_DIS
LIN {X -22.407,Y -139.6216,Z 179,A -94.4774,B 5.4428,C 0.3919,E1 5.4351,E2 186.9211} C_DIS
LIN {X -18.1191,Y -140.2406,Z 179,A -92.7699,B 5.4428,C 0.3929,E1 5.4398,E2 185.2194} C_DIS
LIN {X -14.305,Y -140.6829,Z 179,A -91.3122,B 5.4426,C 0.3944,E1 5.4438,E2 183.7744} C_DIS
LIN {X -11.3424,Y -140.9516,Z 179,A -90.1291,B 5.4426,C 0.3949,E1 5.4471,E2 182.5939} C_DIS
LIN {X -8.3956,Y -141.157,Z 179,A -88.8326,B 5.4426,C 0.3937,E1 5.4507,E2 181.2834} C_DIS
LIN {X -4.8486,Y -141.3246,Z 179,A -87.4885,B 5.4426,C 0.3949,E1 5.4545,E2 179.9515} C_DIS
LIN {X -1.6214,Y -141.3988,Z 179,A -86.1865,B 5.4426,C 0.3949,E1 5.4581,E2 178.6497} C_DIS
LIN {X 0.9995,Y -141.4027,Z 179,A -85.5666,B 5.4422,C 0.4004,E1 5.4597,E2 178.0889} C_DIS
Enddeposition()
LIN {X 0.9995,Y -141.4027,Z 179,A -85.5666,B 5.4422,C 0.4004,E1 5.4597,E2 178.0889} C_DIS
Startdeposition()
$VEL.CP = VEL_PRINT
LIN {X 0.0013,Y -142.3117,Z 179,A -86.0551,B 5.442,C 0.4047,E1 5.4583,E2 178.622} C_DIS
LIN {X -3.2536,Y -142.2741,Z 179,A -87.3393,B 5.442,C 0.4044,E1 5.4547,E2 179.9032} C_DIS
LIN {X -6.9714,Y -142.1387,Z 179,A -88.849,B 5.442,C 0.4046,E1 5.4505,E2 181.4151} C_DIS
LIN {X -10.2874,Y -141.9372,Z 179,A -90.2616,B 5.4419,C 0.4055,E1 5.4465,E2 182.8385} C_DIS
LIN {X -13.715,Y -141.647,Z 179,A -91.6439,B 5.4419,C 0.4052,E1 5.4426,E2 184.2209} C_DIS
LIN {X -17.4145,Y -141.241,Z 179,A -93.096,B 5.4419,C 0.4044,E1 5.4386,E2 185.6674} C_DIS
LIN {X -20.6408,Y -140.8054,Z 179,A -94.4405,B 5.4419,C 0.4044,E1 5.4349,E2 187.0169} C_DIS
LIN {X -24.0878,Y -140.2575,Z 179,A -95.8892,B 5.4419,C 0.4044,E1 5.4309,E2 188.472} C_DIS
LIN {X -27.5336,Y -139.6227,Z 179,A -97.2643,B 5.442,C 0.4035,E1 5.4271,E2 189.8427} C_DIS
LIN {X -31.1724,Y -138.8542,Z 179,A -98.6955,B 5.4422,C 0.4019,E1 5.4232,E2 191.2654} C_DIS
LIN {X -34.3405,Y -138.1054,Z 179,A -100.0865,B 5.4422,C 0.4022,E1 5.4194,E2 192.6676} C_DIS
LIN {X -37.7142,Y -137.2222,Z 179,A -101.497,B 5.4422,C 0.4014,E1 5.4156,E2 194.0793} C_DIS
LIN {X -41.0661,Y -136.2565,Z 179,A -102.8131,B 5.4423,C 0.3994,E1 5.4121,E2 195.3838} C_DIS
LIN {X -44.0813,Y -135.3122,Z 179,A -104.2002,B 5.4423,C 0.3998,E1 5.4084,E2 196.7868} C_DIS
LIN {X -47.664,Y -134.0911,Z 179,A -105.6807,B 5.4424,C 0.3981,E1 5.4045,E2 198.2617} C_DIS
LIN {X -50.8466,Y -132.9176,Z 179,A -107.2088,B 5.4424,C 0.3988,E1 5.4005,E2 199.8119} C_DIS
LIN {X -54.4526,Y -131.4798,Z 179,A -108.6762,B 5.4426,C 0.3961,E1 5.3967,E2 201.2666} C_DIS
LIN {X -57.0544,Y -130.3727,Z 179,A -109.8209,B 5.4426,C 0.395,E1 5.3938,E2 202.4123} C_DIS
LIN {X -60.055,Y -129.0169,Z 179,A -111.1397,B 5.4428,C 0.3935,E1 5.3904,E2 203.7303} C_DIS
LIN {X -63.1952,Y -127.5079,Z 179,A -112.6022,B 5.4428,C 0.3926,E1 5.3867,E2 205.201} C_DIS
LIN {X -66.9099,Y -125.601,Z 179,A -114.288,B 5.443,C 0.3906,E1 5.3825,E2 206.8876} C_DIS
LIN {X -70.5746,Y -123.5785,Z 179,A -116.067,B 5.443,C 0.3895,E1 5.3782,E2 208.6792} C_DIS
LIN {X -74.5508,Y -121.2213,Z 179,A -117.913,B 5.4433,C 0.3868,E1 5.3738,E2 210.5231} C_DIS
LIN {X -78.2396,Y -118.8738,Z 179,A -119.6812,B 5.4434,C 0.3843,E1 5.3696,E2 212.2924} C_DIS
LIN {X -81.8416,Y -116.4234,Z 179,A -121.4617,B 5.4436,C 0.382,E1 5.3655,E2 214.0763} C_DIS
LIN {X -85.3689,Y -113.8629,Z 179,A -123.2727,B 5.4437,C 0.3798,E1 5.3614,E2 215.8948} C_DIS
LIN {X -88.8311,Y -111.1824,Z 179,A -125.0325,B 5.444,C 0.3768,E1 5.3575,E2 217.6539} C_DIS
LIN {X -91.7131,Y -108.8173,Z 179,A -126.6603,B 5.444,C 0.3755,E1 5.354,E2 219.2985} C_DIS
LIN {X -95.0559,Y -105.9094,Z 179,A -128.4538,B 5.4443,C 0.3724,E1 5.3503,E2 221.093} C_DIS
LIN {X -98.2198,Y -102.982,Z 179,A -130.2233,B 5.4444,C 0.3695,E1 5.3466,E2 222.8667} C_DIS
LIN {X -101.3286,Y -99.9254,Z 179,A -132.0311,B 5.4446,C 0.3667,E1 5.3431,E2 224.6811} C_DIS
LIN {X -104.1824,Y -96.9456,Z 179,A -133.6193,B 5.4449,C 0.3626,E1 5.34,E2 226.2592} C_DIS
LIN {X -107.1034,Y -93.7086,Z 179,A -135.4985,B 5.4451,C 0.3603,E1 5.3365,E2 228.1544} C_DIS
LIN {X -109.9378,Y -90.3673,Z 179,A -137.2389,B 5.4453,C 0.3563,E1 5.3334,E2 229.8911} C_DIS
LIN {X -112.6537,Y -86.9576,Z 179,A -138.9989,B 5.4456,C 0.3525,E1 5.3304,E2 231.6512} C_DIS
LIN {X -115.0966,Y -83.6973,Z 179,A -140.7508,B 5.4457,C 0.35,E1 5.3274,E2 233.4174} C_DIS
LIN {X -117.8384,Y -79.7904,Z 179,A -142.6395,B 5.446,C 0.3452,E1 5.3244,E2 235.301} C_DIS
LIN {X -120.1726,Y -76.2303,Z 179,A -144.3929,B 5.4463,C 0.3416,E1 5.3218,E2 237.059} C_DIS
LIN {X -122.0998,Y -73.1036,Z 179,A -146.0034,B 5.4464,C 0.3394,E1 5.3194,E2 238.6863} C_DIS
LIN {X -124.2978,Y -69.301,Z 179,A -147.8188,B 5.4466,C 0.3356,E1 5.3169,E2 240.5072} C_DIS
LIN {X -126.2667,Y -65.6421,Z 179,A -149.4106,B 5.4469,C 0.3306,E1 5.3149,E2 242.0874} C_DIS
LIN {X -127.8379,Y -62.5262,Z 179,A -150.8573,B 5.4471,C 0.3275,E1 5.313,E2 243.5389} C_DIS
LIN {X -129.332,Y -59.3735,Z 179,A -152.2982,B 5.4473,C 0.3243,E1 5.3113,E2 244.9839} C_DIS
LIN {X -131.0985,Y -55.3657,Z 179,A -154.2443,B 5.4475,C 0.3215,E1 5.3092,E2 246.9533} C_DIS
LIN {X -132.6776,Y -51.4639,Z 179,A -155.8588,B 5.4478,C 0.3163,E1 5.3075,E2 248.5562} C_DIS
LIN {X -133.9731,Y -47.9913,Z 179,A -157.3323,B 5.448,C 0.3121,E1 5.3061,E2 250.0264} C_DIS
LIN {X -135.1269,Y -44.6397,Z 179,A -158.8193,B 5.4482,C 0.3089,E1 5.3048,E2 251.5205} C_DIS
LIN {X -136.1803,Y -41.3149,Z 179,A -160.2329,B 5.4484,C 0.3052,E1 5.3036,E2 252.9345} C_DIS
LIN {X -137.1522,Y -37.9648,Z 179,A -161.6992,B 5.4486,C 0.302,E1 5.3025,E2 254.4081} C_DIS
LIN {X -138.0459,Y -34.575,Z 179,A -163.1461,B 5.4488,C 0.2984,E1 5.3015,E2 255.8588} C_DIS
LIN {X -138.8523,Y -31.1805,Z 179,A -164.5681,B 5.449,C 0.2947,E1 5.3006,E2 257.2822} C_DIS
LIN {X -139.5755,Y -27.7666,Z 179,A -166.0032,B 5.4492,C 0.2911,E1 5.2997,E2 258.7203} C_DIS
LIN {X -140.1554,Y -24.669,Z 179,A -167.3535,B 5.4493,C 0.2883,E1 5.2991,E2 260.0804} C_DIS
LIN {X -140.729,Y -21.1587,Z 179,A -168.8307,B 5.4495,C 0.2847,E1 5.2984,E2 261.5626} C_DIS
LIN {X -141.2298,Y -17.5081,Z 179,A -170.272,B 5.4498,C 0.2801,E1 5.2979,E2 262.9973} C_DIS
LIN {X -141.5945,Y -14.2624,Z 179,A -171.7509,B 5.4498,C 0.278,E1 5.2975,E2 264.4967} C_DIS
LIN {X -141.9068,Y -10.7027,Z 179,A -173.1658,B 5.4501,C 0.2737,E1 5.2971,E2 265.9074} C_DIS
LIN {X -142.1373,Y -6.9998,Z 179,A -174.6527,B 5.4503,C 0.2694,E1 5.2969,E2 267.3924} C_DIS
LIN {X -142.2602,Y -3.7521,Z 179,A -176.0518,B 5.4504,C 0.2665,E1 5.2968,E2 268.8023} C_DIS
LIN {X -142.3127,Y -0.0263,Z 179,A -177.572,B 5.4506,C 0.2624,E1 5.2968,E2 270.3241} C_DIS
LIN {X -142.2739,Y 3.258,Z 179,A -179.0164,B 5.4508,C 0.2598,E1 5.2968,E2 271.7832} C_DIS
LIN {X -142.139,Y 6.9665,Z 179,A 179.5748,B 5.451,C 0.2547,E1 5.297,E2 273.1797} C_DIS
LIN {X -141.9261,Y 10.4392,Z 179,A 178.0915,B 5.4512,C 0.2515,E1 5.2973,E2 274.6727} C_DIS
LIN {X -141.6502,Y 13.6816,Z 179,A 176.7152,B 5.4512,C 0.2484,E1 5.2976,E2 276.0565} C_DIS
LIN {X -141.2401,Y 17.4214,Z 179,A 175.2119,B 5.4515,C 0.244,E1 5.2981,E2 277.5571} C_DIS
LIN {X -140.8064,Y 20.634,Z 179,A 173.8412,B 5.4516,C 0.2409,E1 5.2986,E2 278.9353} C_DIS
LIN {X -140.2603,Y 24.071,Z 179,A 172.3728,B 5.4518,C 0.2376,E1 5.2993,E2 280.4113} C_DIS
LIN {X -139.6292,Y 27.5001,Z 179,A 170.9709,B 5.4519,C 0.2336,E1 5.3,E2 281.8118} C_DIS
LIN {X -138.9923,Y 30.5506,Z 179,A 169.6203,B 5.4521,C 0.231,E1 5.3008,E2 283.1737} C_DIS
LIN {X -138.1006,Y 34.3597,Z 179,A 168.0551,B 5.4522,C 0.2266,E1 5.3019,E2 284.7364} C_DIS
LIN {X -137.2163,Y 37.7356,Z 179,A 166.6149,B 5.4524,C 0.223,E1 5.3029,E2 286.1799} C_DIS
LIN {X -136.2499,Y 41.0877,Z 179,A 165.1748,B 5.4525,C 0.2195,E1 5.304,E2 287.6234} C_DIS
LIN {X -135.2017,Y 44.4153,Z 179,A 163.7348,B 5.4527,C 0.216,E1 5.3053,E2 289.0667} C_DIS
LIN {X -134.3224,Y 47.0057,Z 179,A 162.4776,B 5.4527,C 0.2145,E1 5.3064,E2 290.3431} C_DIS
LIN {X -132.8597,Y 50.9955,Z 179,A 160.788,B 5.4529,C 0.2097,E1 5.3081,E2 292.0285} C_DIS
LIN {X -131.4723,Y 54.4705,Z 179,A 159.3104,B 5.4531,C 0.2055,E1 5.3096,E2 293.501} C_DIS
LIN {X -130.1048,Y 57.6612,Z 179,A 158.0144,B 5.4533,C 0.2009,E1 5.3111,E2 294.7828} C_DIS
LIN {X -129.0279,Y 60.0314,Z 179,A 156.8117,B 5.4533,C 0.1996,E1 5.3125,E2 296.0044} C_DIS
LIN {X -127.5237,Y 63.1633,Z 179,A 155.3639,B 5.4534,C 0.1965,E1 5.3143,E2 297.4573} C_DIS
LIN {X -125.9411,Y 66.2622,Z 179,A 153.9574,B 5.4535,C 0.193,E1 5.3161,E2 298.8632} C_DIS
LIN {X -123.8818,Y 70.0418,Z 179,A 152.1389,B 5.4537,C 0.1895,E1 5.3185,E2 300.6913} C_DIS
LIN {X -122.0072,Y 73.2589,Z 179,A 150.4915,B 5.4537,C 0.1872,E1 5.3209,E2 302.3564} C_DIS
LIN {X -119.7047,Y 76.9628,Z 179,A 148.7006,B 5.4539,C 0.1833,E1 5.3236,E2 304.1503} C_DIS
LIN {X -117.3463,Y 80.5125,Z 179,A 146.9382,B 5.4539,C 0.1797,E1 5.3264,E2 305.9171} C_DIS
LIN {X -114.7969,Y 84.1077,Z 179,A 145.1349,B 5.4541,C 0.1759,E1 5.3293,E2 307.7226} C_DIS
LIN {X -112.1107,Y 87.6568,Z 179,A 143.3091,B 5.4542,C 0.1722,E1 5.3324,E2 309.5511} C_DIS
LIN {X -109.3902,Y 91.0292,Z 179,A 141.5027,B 5.4543,C 0.169,E1 5.3356,E2 311.3639} C_DIS
LIN {X -106.6432,Y 94.2319,Z 179,A 139.7813,B 5.4544,C 0.1656,E1 5.3388,E2 313.0867} C_DIS
LIN {X -103.7108,Y 97.4503,Z 179,A 138.114,B 5.4546,C 0.1611,E1 5.3419,E2 314.7416} C_DIS
LIN {X -100.9366,Y 100.3205,Z 179,A 136.4035,B 5.4546,C 0.1589,E1 5.3453,E2 316.4639} C_DIS
LIN {X -97.5115,Y 103.653,Z 179,A 134.5061,B 5.4547,C 0.1548,E1 5.3491,E2 318.3563} C_DIS
LIN {X -94.3816,Y 106.5108,Z 179,A 132.758,B 5.4548,C 0.152,E1 5.3528,E2 320.1083} C_DIS
LIN {X -91.0469,Y 109.3755,Z 179,A 130.9398,B 5.4549,C 0.1493,E1 5.3566,E2 321.9312} C_DIS
LIN {X -87.6648,Y 112.1044,Z 179,A 129.1772,B 5.4549,C 0.1463,E1 5.3605,E2 323.694} C_DIS
LIN {X -84.1977,Y 114.7308,Z 179,A 127.3918,B 5.4551,C 0.1437,E1 5.3645,E2 325.4824} C_DIS
LIN {X -80.6695,Y 117.2385,Z 179,A 125.6003,B 5.4551,C 0.1414,E1 5.3686,E2 327.2787} C_DIS
LIN {X -76.9667,Y 119.7022,Z 179,A 123.8204,B 5.4551,C 0.1386,E1 5.3727,E2 329.0559} C_DIS
LIN {X -73.2622,Y 122.0052,Z 179,A 121.9695,B 5.4552,C 0.137,E1 5.3772,E2 330.9174} C_DIS
LIN {X -69.2836,Y 124.3075,Z 179,A 120.0633,B 5.4552,C 0.135,E1 5.3818,E2 332.8293} C_DIS
LIN {X -65.6496,Y 126.2628,Z 179,A 118.5003,B 5.4554,C 0.1318,E1 5.3857,E2 334.3785} C_DIS
LIN {X -62.5152,Y 127.8434,Z 179,A 117.0545,B 5.4554,C 0.1304,E1 5.3893,E2 335.8274} C_DIS
LIN {X -58.4677,Y 129.7441,Z 179,A 115.1327,B 5.4554,C 0.1296,E1 5.3942,E2 337.7633} C_DIS
LIN {X -54.6857,Y 131.3825,Z 179,A 113.5793,B 5.4554,C 0.1267,E1 5.3981,E2 339.3021} C_DIS
LIN {X -51.4522,Y 132.6821,Z 179,A 112.1305,B 5.4554,C 0.1257,E1 5.4019,E2 340.7557} C_DIS
LIN {X -47.9746,Y 133.9791,Z 179,A 110.6826,B 5.4555,C 0.1238,E1 5.4057,E2 342.1967} C_DIS
LIN {X -44.64,Y 135.1268,Z 179,A 109.2244,B 5.4555,C 0.123,E1 5.4096,E2 343.6589} C_DIS
LIN {X -41.3149,Y 136.1803,Z 179,A 107.8533,B 5.4555,C 0.1215,E1 5.4132,E2 345.0248} C_DIS
LIN {X -37.9382,Y 137.1596,Z 179,A 106.3849,B 5.4555,C 0.121,E1 5.4172,E2 346.4991} C_DIS
LIN {X -34.5656,Y 138.0483,Z 179,A 104.9853,B 5.4556,C 0.12,E1 5.421,E2 347.8972} C_DIS
LIN {X -31.1915,Y 138.8498,Z 179,A 103.5903,B 5.4556,C 0.1192,E1 5.4248,E2 349.2912} C_DIS
LIN {X -27.7949,Y 139.5698,Z 179,A 102.1692,B 5.4556,C 0.1187,E1 5.4286,E2 350.7145} C_DIS
LIN {X -24.6018,Y 140.1674,Z 179,A 100.8405,B 5.4556,C 0.1183,E1 5.4323,E2 352.0451} C_DIS
LIN {X -21.159,Y 140.7289,Z 179,A 99.3927,B 5.4556,C 0.1183,E1 5.4363,E2 353.4976} C_DIS
LIN {X -17.4238,Y 141.2399,Z 179,A 97.977,B 5.4556,C 0.1166,E1 5.4402,E2 354.8996} C_DIS
LIN {X -14.1899,Y 141.6014,Z 179,A 96.5347,B 5.4556,C 0.1178,E1 5.4442,E2 356.3579} C_DIS
LIN {X -10.7169,Y 141.9058,Z 179,A 95.1883,B 5.4556,C 0.1168,E1 5.448,E2 357.6963} C_DIS
LIN {X -6.3461,Y 142.1701,Z 179,A 93.2359,B 5.4556,C 0.1189,E1 5.4535,E2 359.672} C_DIS
LIN {X -1.7502,Y 142.3001,Z 179,A 91.602,B 5.4557,C 0.1162,E1 5.458,E2 361.2776} C_DIS
LIN {X 1.5054,Y 142.3034,Z 179,A 90.2661,B 5.4557,C 0.1166,E1 5.4617,E2 362.6161} C_DIS
LIN {X 5.2226,Y 142.214,Z 179,A 88.7658,B 5.4557,C 0.1168,E1 5.4659,E2 364.1161} C_DIS
LIN {X 8.4951,Y 142.0559,Z 179,A 87.4098,B 5.4557,C 0.1176,E1 5.4697,E2 365.4762} C_DIS
LIN {X 12.206,Y 141.7852,Z 179,A 85.9986,B 5.4557,C 0.1169,E1 5.4736,E2 366.8758} C_DIS
LIN {X 15.6765,Y 141.444,Z 179,A 84.5729,B 5.4557,C 0.1176,E1 5.4776,E2 368.3038} C_DIS
LIN {X 18.9078,Y 141.0483,Z 179,A 83.2647,B 5.4557,C 0.1181,E1 5.4812,E2 369.6112} C_DIS
LIN {X 22.2234,Y 140.5641,Z 179,A 81.9103,B 5.4557,C 0.1188,E1 5.4849,E2 370.9658} C_DIS
LIN {X 26.0446,Y 139.9074,Z 179,A 80.425,B 5.4557,C 0.1187,E1 5.489,E2 372.4411} C_DIS
LIN {X 29.237,Y 139.2759,Z 179,A 78.9834,B 5.4556,C 0.1212,E1 5.493,E2 373.8991} C_DIS
LIN {X 32.6401,Y 138.5174,Z 179,A 77.6573,B 5.4556,C 0.1212,E1 5.4966,E2 375.215} C_DIS
LIN {X 36.0242,Y 137.6757,Z 179,A 76.2658,B 5.4556,C 0.122,E1 5.5003,E2 376.6045} C_DIS
LIN {X 39.4151,Y 136.7432,Z 179,A 74.7582,B 5.4556,C 0.1243,E1 5.5044,E2 378.1235} C_DIS
LIN {X 43.8017,Y 135.4015,Z 179,A 73.031,B 5.4556,C 0.1243,E1 5.509,E2 379.835} C_DIS
LIN {X 47.638,Y 134.1005,Z 179,A 71.4861,B 5.4556,C 0.1248,E1 5.513,E2 381.3686} C_DIS
LIN {X 50.9929,Y 132.8607,Z 179,A 69.9273,B 5.4554,C 0.1279,E1 5.5171,E2 382.9425} C_DIS
LIN {X 53.9406,Y 131.6924,Z 179,A 68.5907,B 5.4554,C 0.1301,E1 5.5206,E2 384.2866} C_DIS
LIN {X 57.669,Y 130.1014,Z 179,A 67.2488,B 5.4554,C 0.1281,E1 5.524,E2 385.5912} C_DIS
LIN {X 60.7332,Y 128.7003,Z 179,A 65.7397,B 5.4554,C 0.1318,E1 5.5278,E2 387.1197} C_DIS
LIN {X 63.9745,Y 127.1202,Z 179,A 64.3479,B 5.4554,C 0.1329,E1 5.5313,E2 388.5038} C_DIS
LIN {X 67.1447,Y 125.4754,Z 179,A 62.7999,B 5.4552,C 0.1363,E1 5.5351,E2 390.0658} C_DIS
LIN {X 70.8999,Y 123.3929,Z 179,A 61.1813,B 5.4552,C 0.1373,E1 5.5391,E2 391.6703} C_DIS
LIN {X 74.558,Y 121.217,Z 179,A 59.5157,B 5.4552,C 0.1392,E1 5.543,E2 393.3298} C_DIS
LIN {X 77.6031,Y 119.2903,Z 179,A 58.0861,B 5.4552,C 0.1411,E1 5.5464,E2 394.7567} C_DIS
LIN {X 81.1239,Y 116.9246,Z 179,A 56.4089,B 5.4551,C 0.1435,E1 5.5502,E2 396.4301} C_DIS
LIN {X 84.1534,Y 114.7634,Z 179,A 54.8281,B 5.455,C 0.1472,E1 5.5538,E2 398.0216} C_DIS
LIN {X 87.6478,Y 112.1177,Z 179,A 53.0774,B 5.4549,C 0.1501,E1 5.5577,E2 399.7707} C_DIS
LIN {X 90.9518,Y 109.4543,Z 179,A 51.5075,B 5.4549,C 0.1512,E1 5.5611,E2 401.323} C_DIS
LIN {X 93.7306,Y 107.0842,Z 179,A 50.0939,B 5.4548,C 0.1532,E1 5.564,E2 402.7295} C_DIS
LIN {X 96.7429,Y 104.3711,Z 179,A 48.4195,B 5.4547,C 0.1569,E1 5.5675,E2 404.4097} C_DIS
LIN {X 99.8855,Y 101.3677,Z 179,A 46.6988,B 5.4546,C 0.16,E1 5.571,E2 406.1269} C_DIS
LIN {X 102.9847,Y 98.217,Z 179,A 44.9982,B 5.4546,C 0.1625,E1 5.5743,E2 407.8178} C_DIS
LIN {X 105.5189,Y 95.4893,Z 179,A 43.4165,B 5.4544,C 0.1669,E1 5.5773,E2 409.4105} C_DIS
LIN {X 108.3158,Y 92.3045,Z 179,A 41.7396,B 5.4543,C 0.1701,E1 5.5803,E2 411.0841} C_DIS
LIN {X 111.15,Y 88.8718,Z 179,A 39.9796,B 5.4542,C 0.1736,E1 5.5834,E2 412.8404} C_DIS
LIN {X 113.8541,Y 85.3806,Z 179,A 38.2174,B 5.4541,C 0.1774,E1 5.5864,E2 414.6013} C_DIS
LIN {X 116.4247,Y 81.8398,Z 179,A 36.5003,B 5.4539,C 0.1809,E1 5.5892,E2 416.3133} C_DIS
LIN {X 118.876,Y 78.2362,Z 179,A 34.8152,B 5.4539,C 0.184,E1 5.5918,E2 417.9899} C_DIS
LIN {X 121.1547,Y 74.6595,Z 179,A 33.2273,B 5.4538,C 0.1863,E1 5.5941,E2 419.563} C_DIS
LIN {X 123.3262,Y 71.0153,Z 179,A 31.5427,B 5.4536,C 0.1902,E1 5.5965,E2 421.2454} C_DIS
LIN {X 125.4521,Y 67.1879,Z 179,A 29.8269,B 5.4536,C 0.1939,E1 5.5988,E2 422.9558} C_DIS
LIN {X 127.068,Y 64.0769,Z 179,A 28.4715,B 5.4534,C 0.1966,E1 5.6005,E2 424.3046} C_DIS
LIN {X 128.6493,Y 60.84,Z 179,A 27.0972,B 5.4534,C 0.1992,E1 5.6021,E2 425.6697} C_DIS
LIN {X 130.1002,Y 57.6716,Z 179,A 25.5513,B 5.4531,C 0.205,E1 5.6039,E2 427.2349} C_DIS
LIN {X 132.0431,Y 53.0708,Z 179,A 23.7267,B 5.4531,C 0.2074,E1 5.6059,E2 429.0363} C_DIS
LIN {X 133.3077,Y 49.809,Z 179,A 22.3194,B 5.4529,C 0.2111,E1 5.6073,E2 430.4442} C_DIS
LIN {X 134.4923,Y 46.5156,Z 179,A 20.9459,B 5.4527,C 0.2144,E1 5.6085,E2 431.8139} C_DIS
LIN {X 135.6635,Y 42.9814,Z 179,A 19.5158,B 5.4527,C 0.2174,E1 5.6097,E2 433.2359} C_DIS
LIN {X 136.6504,Y 39.7319,Z 179,A 18.2118,B 5.4525,C 0.2201,E1 5.6108,E2 434.5324} C_DIS
LIN {X 137.6157,Y 36.2492,Z 179,A 16.7652,B 5.4524,C 0.224,E1 5.6118,E2 435.9788} C_DIS
LIN {X 138.4632,Y 32.8649,Z 179,A 15.3976,B 5.4522,C 0.2273,E1 5.6127,E2 437.3425} C_DIS
LIN {X 139.1772,Y 29.6944,Z 179,A 14.1238,B 5.4521,C 0.2304,E1 5.6135,E2 438.6126} C_DIS
LIN {X 139.9067,Y 26.0482,Z 179,A 12.6757,B 5.4519,C 0.2338,E1 5.6143,E2 440.0552} C_DIS
LIN {X 140.5034,Y 22.6142,Z 179,A 11.3049,B 5.4518,C 0.2372,E1 5.6149,E2 441.4227} C_DIS
LIN {X 141.0143,Y 19.1671,Z 179,A 9.9123,B 5.4516,C 0.241,E1 5.6155,E2 442.815} C_DIS
LIN {X 141.4177,Y 15.9214,Z 179,A 8.6242,B 5.4515,C 0.2443,E1 5.6159,E2 444.1002} C_DIS
LIN {X 141.7849,Y 12.2094,Z 179,A 7.2249,B 5.4514,C 0.247,E1 5.6162,E2 445.487} C_DIS
LIN {X 141.9919,Y 9.5348,Z 179,A 5.9456,B 5.4511,C 0.2532,E1 5.6165,E2 446.7934} C_DIS
LIN {X 142.2039,Y 5.482,Z 179,A 4.537,B 5.4511,C 0.2543,E1 5.6167,E2 448.1735} C_DIS
LIN {X 142.3003,Y 1.7407,Z 179,A 3.1176,B 5.4509,C 0.2572,E1 5.6167,E2 449.5826} C_DIS
LIN {X 142.3036,Y -1.4815,Z 179,A 1.792,B 5.4507,C 0.2614,E1 5.6167,E2 450.9129} C_DIS
LIN {X 142.2136,Y -5.233,Z 179,A 0.3212,B 5.4505,C 0.265,E1 5.6167,E2 452.3795} C_DIS
LIN {X 142.0566,Y -8.4838,Z 179,A -0.9943,B 5.4503,C 0.2688,E1 5.6164,E2 453.6968} C_DIS
LIN {X 141.8391,Y -11.5676,Z 179,A -2.246,B 5.4502,C 0.2725,E1 5.6161,E2 454.9504} C_DIS
LIN {X 141.4428,Y -15.6881,Z 179,A -3.7747,B 5.45,C 0.2751,E1 5.6157,E2 456.4622} C_DIS
LIN {X 141.0471,Y -18.9169,Z 179,A -5.0532,B 5.4499,C 0.2783,E1 5.6152,E2 457.7376} C_DIS
LIN {X 140.5058,Y -22.5992,Z 179,A -6.5055,B 5.4497,C 0.2818,E1 5.6146,E2 459.1851} C_DIS
LIN {X 139.9093,Y -26.0346,Z 179,A -7.8298,B 5.4495,C 0.2845,E1 5.614,E2 460.5} C_DIS
LIN {X 139.2733,Y -29.2489,Z 179,A -9.1507,B 5.4493,C 0.2882,E1 5.6133,E2 461.8223} C_DIS
LIN {X 138.5157,Y -32.647,Z 179,A -10.5456,B 5.4491,C 0.292,E1 5.6124,E2 463.2175} C_DIS
LIN {X 137.6754,Y -36.0252,Z 179,A -11.9105,B 5.449,C 0.2954,E1 5.6114,E2 464.5786} C_DIS
LIN {X 136.9093,Y -38.8331,Z 179,A -13.1417,B 5.4487,C 0.2995,E1 5.6105,E2 465.8187} C_DIS
LIN {X 135.7467,Y -42.7211,Z 179,A -14.5543,B 5.4487,C 0.3005,E1 5.6094,E2 467.2032} C_DIS
LIN {X 134.6444,Y -46.0768,Z 179,A -16.093,B 5.4484,C 0.3062,E1 5.608,E2 468.7588} C_DIS
LIN {X 133.4705,Y -49.3742,Z 179,A -17.4038,B 5.4482,C 0.3085,E1 5.6068,E2 470.0577} C_DIS
LIN {X 132.1325,Y -52.8489,Z 179,A -18.8663,B 5.448,C 0.312,E1 5.6053,E2 471.5167} C_DIS
LIN {X 130.7985,Y -56.0697,Z 179,A -20.2352,B 5.4479,C 0.3152,E1 5.6038,E2 472.8821} C_DIS
LIN {X 129.7461,Y -58.4631,Z 179,A -21.2689,B 5.4477,C 0.3176,E1 5.6026,E2 473.9143} C_DIS
LIN {X 128.3253,Y -61.5181,Z 179,A -22.6078,B 5.4475,C 0.3209,E1 5.601,E2 475.252} C_DIS
LIN {X 126.7268,Y -64.7472,Z 179,A -24.0093,B 5.4473,C 0.3239,E1 5.5993,E2 476.6482} C_DIS
LIN {X 125.0368,Y -67.9578,Z 179,A -25.5386,B 5.4471,C 0.3287,E1 5.5973,E2 478.1881} C_DIS
LIN {X 122.9543,Y -71.6577,Z 179,A -27.1294,B 5.4469,C 0.3311,E1 5.5951,E2 479.7645} C_DIS
LIN {X 120.7504,Y -75.3111,Z 179,A -28.8175,B 5.4467,C 0.3349,E1 5.5926,E2 481.4502} C_DIS
LIN {X 118.3935,Y -78.9645,Z 179,A -30.5152,B 5.4465,C 0.3384,E1 5.59,E2 483.1424} C_DIS
LIN {X 115.9258,Y -82.5452,Z 179,A -32.2535,B 5.4462,C 0.3424,E1 5.5872,E2 484.8806} C_DIS
LIN {X 113.3466,Y -86.0531,Z 179,A -33.9679,B 5.446,C 0.3459,E1 5.5844,E2 486.5914} C_DIS
LIN {X 110.6331,Y -89.5141,Z 179,A -35.6774,B 5.4458,C 0.349,E1 5.5814,E2 488.2943} C_DIS
LIN {X 108.3314,Y -92.2862,Z 179,A -37.099,B 5.4456,C 0.3518,E1 5.5789,E2 489.7133} C_DIS
LIN {X 105.5328,Y -95.474,Z 179,A -38.7483,B 5.4454,C 0.3547,E1 5.5758,E2 491.3562} C_DIS
LIN {X 103.161,Y -98.0326,Z 179,A -40.0142,B 5.4454,C 0.3556,E1 5.5734,E2 492.6047} C_DIS
LIN {X 101.1619,Y -100.0937,Z 179,A -41.2229,B 5.4452,C 0.3588,E1 5.5711,E2 493.8215} C_DIS
LIN {X 98.6044,Y -102.6145,Z 179,A -42.7873,B 5.4448,C 0.3636,E1 5.5679,E2 495.4032} C_DIS
LIN {X 95.5783,Y -105.4381,Z 179,A -44.4483,B 5.4446,C 0.3668,E1 5.5645,E2 497.0648} C_DIS
LIN {X 92.3764,Y -108.2547,Z 179,A -45.9995,B 5.4446,C 0.3677,E1 5.5613,E2 498.5952} C_DIS
LIN {X 89.5146,Y -110.6327,Z 179,A -47.5848,B 5.4443,C 0.3718,E1 5.5578,E2 500.1935} C_DIS
LIN {X 86.2707,Y -113.1805,Z 179,A -49.1298,B 5.4443,C 0.3732,E1 5.5544,E2 501.7244} C_DIS
LIN {X 83.2817,Y -115.3978,Z 179,A -50.7221,B 5.4439,C 0.3772,E1 5.5508,E2 503.3305} C_DIS
LIN {X 79.7851,Y -117.8421,Z 179,A -52.2956,B 5.4439,C 0.378,E1 5.5472,E2 504.8861} C_DIS
LIN {X 76.2435,Y -120.1643,Z 179,A -54.0027,B 5.4437,C 0.3808,E1 5.5432,E2 506.5948} C_DIS
LIN {X 72.5317,Y -122.4407,Z 179,A -55.6879,B 5.4435,C 0.3826,E1 5.5392,E2 508.2722} C_DIS
LIN {X 69.4106,Y -124.2366,Z 179,A -57.1721,B 5.4434,C 0.3853,E1 5.5356,E2 509.7622} C_DIS
LIN {X 65.6466,Y -126.2644,Z 179,A -58.8188,B 5.4433,C 0.3867,E1 5.5315,E2 511.4002} C_DIS
LIN {X 62.5159,Y -127.843,Z 179,A -60.2191,B 5.4431,C 0.3885,E1 5.528,E2 512.8} C_DIS
LIN {X 59.364,Y -129.3365,Z 179,A -61.5959,B 5.4431,C 0.3899,E1 5.5246,E2 514.1742} C_DIS
LIN {X 56.2843,Y -130.7057,Z 179,A -62.9355,B 5.4429,C 0.3914,E1 5.5211,E2 515.5124} C_DIS
LIN {X 53.0645,Y -132.0456,Z 179,A -64.3236,B 5.4429,C 0.3928,E1 5.5175,E2 516.8994} C_DIS
LIN {X 49.5948,Y -133.3879,Z 179,A -65.8064,B 5.4427,C 0.3943,E1 5.5137,E2 518.3812} C_DIS
LIN {X 46.5301,Y -134.4873,Z 179,A -67.1362,B 5.4426,C 0.3959,E1 5.5102,E2 519.7145} C_DIS
LIN {X 42.9773,Y -135.6648,Z 179,A -68.5993,B 5.4426,C 0.3968,E1 5.5063,E2 521.1726} C_DIS
LIN {X 39.62,Y -136.6832,Z 179,A -69.9951,B 5.4425,C 0.3979,E1 5.5026,E2 522.5672} C_DIS
LIN {X 36.3795,Y -137.581,Z 179,A -71.3489,B 5.4424,C 0.3991,E1 5.4989,E2 523.9218} C_DIS
LIN {X 32.9082,Y -138.4528,Z 179,A -72.7665,B 5.4424,C 0.3999,E1 5.4951,E2 525.3372} C_DIS
LIN {X 29.7041,Y -139.175,Z 179,A -74.1009,B 5.4422,C 0.401,E1 5.4914,E2 526.674} C_DIS
LIN {X 26.0592,Y -139.9046,Z 179,A -75.5537,B 5.4422,C 0.4014,E1 5.4874,E2 528.1219} C_DIS
LIN {X 22.6243,Y -140.5017,Z 179,A -76.9532,B 5.4422,C 0.4022,E1 5.4836,E2 529.5217} C_DIS
LIN {X 19.1773,Y -141.013,Z 179,A -78.3001,B 5.4422,C 0.4022,E1 5.4799,E2 530.8618} C_DIS
LIN {X 15.9194,Y -141.4179,Z 179,A -79.6943,B 5.442,C 0.4038,E1 5.476,E2 532.2665} C_DIS
LIN {X 12.2162,Y -141.7843,Z 179,A -81.1241,B 5.442,C 0.4034,E1 5.472,E2 533.6879} C_DIS
LIN {X 8.9701,Y -142.0267,Z 179,A -82.523,B 5.442,C 0.405,E1 5.4681,E2 535.0994} C_DIS
LIN {X 5.4862,Y -142.2037,Z 179,A -83.8516,B 5.442,C 0.4044,E1 5.4644,E2 536.4184} C_DIS
LIN {X 1.7461,Y -142.3002,Z 179,A -85.3629,B 5.442,C 0.4047,E1 5.4602,E2 537.9311} C_DIS
LIN {X 1.7461,Y -142.3002,Z 179,A -85.3629,B 5.442,C 0.4047,E1 5.4602,E2 537.9311} C_DIS
Enddeposition()
LIN {X 0.9654,Y -133.3724,Z 180,A -85.8777,B 5.8272,C 0.3801,E1 5.8426,E2 538.0345} C_DIS
Startdeposition()
$VEL.CP = VEL_PRINT
LIN {X 3.3739,Y -133.3344,Z 180,A -84.5218,B 5.8274,C 0.3758,E1 5.8465,E2 536.6377} C_DIS
LIN {X 6.6395,Y -133.2112,Z 180,A -83.1236,B 5.8274,C 0.3755,E1 5.8504,E2 535.2395} C_DIS
LIN {X 9.8994,Y -133.0088,Z 180,A -81.7117,B 5.8274,C 0.3749,E1 5.8544,E2 533.8257} C_DIS
LIN {X 13.1794,Y -132.7245,Z 180,A -80.3072,B 5.8275,C 0.3745,E1 5.8583,E2 532.4217} C_DIS
LIN {X 16.4281,Y -132.3624,Z 180,A -78.911,B 5.8275,C 0.374,E1 5.8621,E2 531.0259} C_DIS
LIN {X 19.8758,Y -131.8882,Z 180,A -77.4721,B 5.8275,C 0.374,E1 5.8661,E2 529.593} C_DIS
LIN {X 22.7907,Y -131.4167,Z 180,A -76.1366,B 5.8277,C 0.3723,E1 5.8698,E2 528.2484} C_DIS
LIN {X 26.0241,Y -130.8141,Z 180,A -74.7058,B 5.8277,C 0.3711,E1 5.8737,E2 526.8145} C_DIS
LIN {X 29.3235,Y -130.1135,Z 180,A -73.3281,B 5.8277,C 0.3711,E1 5.8775,E2 525.4448} C_DIS
LIN {X 32.4067,Y -129.3801,Z 180,A -71.9208,B 5.8279,C 0.3693,E1 5.8813,E2 524.0309} C_DIS
LIN {X 35.668,Y -128.5188,Z 180,A -70.5376,B 5.8279,C 0.3689,E1 5.885,E2 522.655} C_DIS
LIN {X 38.7153,Y -127.6341,Z 180,A -69.1578,B 5.8279,C 0.3674,E1 5.8887,E2 521.2722} C_DIS
LIN {X 42.312,Y -126.4869,Z 180,A -67.6258,B 5.8279,C 0.3671,E1 5.8928,E2 519.7503} C_DIS
LIN {X 44.9374,Y -125.5784,Z 180,A -66.3713,B 5.8281,C 0.365,E1 5.8961,E2 518.4873} C_DIS
LIN {X 48.0931,Y -124.4038,Z 180,A -64.9393,B 5.8282,C 0.3635,E1 5.8998,E2 517.0561} C_DIS
LIN {X 51.0267,Y -123.23,Z 180,A -63.5915,B 5.8283,C 0.3621,E1 5.9033,E2 515.7086} C_DIS
LIN {X 54.0487,Y -121.9349,Z 180,A -62.1803,B 5.8284,C 0.3603,E1 5.9069,E2 514.2964} C_DIS
LIN {X 57.0215,Y -120.5736,Z 180,A -60.8137,B 5.8284,C 0.359,E1 5.9104,E2 512.9336} C_DIS
LIN {X 59.959,Y -119.1405,Z 180,A -59.428,B 5.8286,C 0.3574,E1 5.9138,E2 511.5491} C_DIS
LIN {X 62.8597,Y -117.637,Z 180,A -57.9024,B 5.8288,C 0.3536,E1 5.9177,E2 510.007} C_DIS
LIN {X 66.3547,Y -115.7016,Z 180,A -56.484,B 5.8288,C 0.3553,E1 5.921,E2 508.6248} C_DIS
LIN {X 68.6664,Y -114.3451,Z 180,A -55.2124,B 5.8289,C 0.3518,E1 5.9241,E2 507.3372} C_DIS
LIN {X 71.3609,Y -112.6826,Z 180,A -53.8452,B 5.8291,C 0.3495,E1 5.9274,E2 505.968} C_DIS
LIN {X 74.1887,Y -110.8412,Z 180,A -52.3309,B 5.8293,C 0.3461,E1 5.9309,E2 504.4443} C_DIS
LIN {X 76.8843,Y -108.9886,Z 180,A -51.0734,B 5.8293,C 0.3459,E1 5.9337,E2 503.2042} C_DIS
LIN {X 79.4505,Y -107.1326,Z 180,A -49.6999,B 5.8294,C 0.3433,E1 5.9368,E2 501.828} C_DIS
LIN {X 82.7046,Y -104.6414,Z 180,A -47.8254,B 5.8297,C 0.3383,E1 5.941,E2 499.9376} C_DIS
LIN {X 85.8716,Y -102.0578,Z 180,A -46.2476,B 5.8297,C 0.3376,E1 5.9444,E2 498.3807} C_DIS
LIN {X 88.9197,Y -99.4133,Z 180,A -44.5267,B 5.83,C 0.3344,E1 5.948,E2 496.6598} C_DIS
LIN {X 91.9232,Y -96.6433,Z 180,A -42.8104,B 5.8301,C 0.3315,E1 5.9515,E2 494.9469} C_DIS
LIN {X 94.3498,Y -94.276,Z 180,A -41.251,B 5.8304,C 0.3269,E1 5.9546,E2 493.3732} C_DIS
LIN {X 97.1934,Y -91.3412,Z 180,A -39.5198,B 5.8306,C 0.3235,E1 5.9579,E2 491.6436} C_DIS
LIN {X 99.9459,Y -88.3206,Z 180,A -37.8042,B 5.8307,C 0.3202,E1 5.9611,E2 489.9313} C_DIS
LIN {X 103.0704,Y -84.654,Z 180,A -35.908,B 5.8309,C 0.3182,E1 5.9645,E2 488.0551} C_DIS
LIN {X 105.6159,Y -81.4561,Z 180,A -34.2104,B 5.831,C 0.3151,E1 5.9674,E2 486.3632} C_DIS
LIN {X 107.1891,Y -79.3745,Z 180,A -33.1038,B 5.8312,C 0.3127,E1 5.9692,E2 485.2574} C_DIS
LIN {X 109.1095,Y -76.7128,Z 180,A -31.7287,B 5.8313,C 0.3098,E1 5.9715,E2 483.8854} C_DIS
LIN {X 110.9011,Y -74.099,Z 180,A -30.3617,B 5.8315,C 0.3065,E1 5.9736,E2 482.5164} C_DIS
LIN {X 112.7404,Y -71.2693,Z 180,A -28.9888,B 5.8316,C 0.3041,E1 5.9757,E2 481.1518} C_DIS
LIN {X 114.4542,Y -68.4835,Z 180,A -27.5905,B 5.8318,C 0.3007,E1 5.9777,E2 479.7531} C_DIS
LIN {X 116.4675,Y -65.0015,Z 180,A -25.9441,B 5.8319,C 0.2976,E1 5.9799,E2 478.1153} C_DIS
LIN {X 117.6868,Y -62.7671,Z 180,A -24.8135,B 5.8321,C 0.2942,E1 5.9814,E2 476.9791} C_DIS
LIN {X 119.1877,Y -59.8662,Z 180,A -23.4472,B 5.8323,C 0.2912,E1 5.9832,E2 475.6161} C_DIS
LIN {X 120.6185,Y -56.9276,Z 180,A -22.0764,B 5.8324,C 0.288,E1 5.9848,E2 474.2481} C_DIS
LIN {X 121.9773,Y -53.9539,Z 180,A -20.7023,B 5.8326,C 0.2848,E1 5.9864,E2 472.8765} C_DIS
LIN {X 123.2233,Y -51.0426,Z 180,A -19.3775,B 5.8327,C 0.2817,E1 5.9878,E2 471.5549} C_DIS
LIN {X 124.5266,Y -47.7772,Z 180,A -17.9098,B 5.8329,C 0.2783,E1 5.9893,E2 470.0912} C_DIS
LIN {X 125.5789,Y -44.9359,Z 180,A -16.632,B 5.833,C 0.2752,E1 5.9905,E2 468.8152} C_DIS
LIN {X 126.6741,Y -41.7499,Z 180,A -15.0799,B 5.8333,C 0.2696,E1 5.9919,E2 467.2487} C_DIS
LIN {X 128.1138,Y -37.0976,Z 180,A -13.2164,B 5.8333,C 0.2674,E1 5.9934,E2 465.4118} C_DIS
LIN {X 129,Y -33.8892,Z 180,A -11.7829,B 5.8336,C 0.2634,E1 5.9944,E2 463.9766} C_DIS
LIN {X 129.7686,Y -30.8148,Z 180,A -10.455,B 5.8337,C 0.2601,E1 5.9953,E2 462.6517} C_DIS
LIN {X 130.5076,Y -27.5213,Z 180,A -9.043,B 5.8339,C 0.2566,E1 5.9962,E2 461.2432} C_DIS
LIN {X 131.1433,Y -24.3153,Z 180,A -7.6768,B 5.834,C 0.2533,E1 5.9969,E2 459.8805} C_DIS
LIN {X 131.702,Y -21.0789,Z 180,A -6.3123,B 5.8342,C 0.25,E1 5.9975,E2 458.5205} C_DIS
LIN {X 132.1648,Y -17.9479,Z 180,A -4.9498,B 5.8343,C 0.2461,E1 5.998,E2 457.1566} C_DIS
LIN {X 132.5644,Y -14.7023,Z 180,A -3.5818,B 5.8345,C 0.2427,E1 5.9985,E2 455.7919} C_DIS
LIN {X 132.8846,Y -11.4471,Z 180,A -2.1954,B 5.8346,C 0.239,E1 5.9988,E2 454.4066} C_DIS
LIN {X 133.1252,Y -8.1852,Z 180,A -0.7963,B 5.8348,C 0.235,E1 5.9991,E2 453.0071} C_DIS
LIN {X 133.2866,Y -4.9066,Z 180,A 0.5243,B 5.8348,C 0.2324,E1 5.9992,E2 451.6965} C_DIS
LIN {X 133.3724,Y -1.1957,Z 180,A 1.8914,B 5.8349,C 0.2314,E1 5.9993,E2 450.3563} C_DIS
LIN {X 133.368,Y 1.6301,Z 180,A 3.3122,B 5.8352,C 0.2247,E1 5.9993,E2 448.909} C_DIS
LIN {X 133.2869,Y 4.8996,Z 180,A 4.6703,B 5.8353,C 0.2214,E1 5.9992,E2 447.5556} C_DIS
LIN {X 133.1254,Y 8.1814,Z 180,A 6.0311,B 5.8354,C 0.2182,E1 5.9989,E2 446.2} C_DIS
LIN {X 132.8762,Y 11.5465,Z 180,A 7.4212,B 5.8356,C 0.215,E1 5.9986,E2 444.8161} C_DIS
LIN {X 132.5539,Y 14.7998,Z 180,A 8.7882,B 5.8356,C 0.2116,E1 5.9982,E2 443.4527} C_DIS
LIN {X 132.1524,Y 18.0427,Z 180,A 10.1552,B 5.8358,C 0.2082,E1 5.9977,E2 442.0893} C_DIS
LIN {X 131.6673,Y 21.2937,Z 180,A 11.5227,B 5.8359,C 0.2049,E1 5.9972,E2 440.7262} C_DIS
LIN {X 131.1246,Y 24.4133,Z 180,A 12.8852,B 5.8361,C 0.2011,E1 5.9965,E2 439.3625} C_DIS
LIN {X 130.4641,Y 27.7226,Z 180,A 14.2959,B 5.8361,C 0.1976,E1 5.9957,E2 437.9555} C_DIS
LIN {X 129.7669,Y 30.8219,Z 180,A 15.6277,B 5.8363,C 0.1944,E1 5.9949,E2 436.6269} C_DIS
LIN {X 128.9447,Y 34.0966,Z 180,A 17.042,B 5.8363,C 0.1909,E1 5.9939,E2 435.2161} C_DIS
LIN {X 128.0986,Y 37.1496,Z 180,A 18.3705,B 5.8365,C 0.1877,E1 5.9929,E2 433.8907} C_DIS
LIN {X 127.1434,Y 40.297,Z 180,A 19.7729,B 5.8366,C 0.184,E1 5.9917,E2 432.4888} C_DIS
LIN {X 126.0505,Y 43.5947,Z 180,A 21.1519,B 5.8366,C 0.1817,E1 5.9905,E2 431.1227} C_DIS
LIN {X 125.0264,Y 46.4512,Z 180,A 22.5026,B 5.8368,C 0.1775,E1 5.9892,E2 429.7655} C_DIS
LIN {X 123.8248,Y 49.5651,Z 180,A 23.8431,B 5.8368,C 0.1751,E1 5.9878,E2 428.4356} C_DIS
LIN {X 122.5877,Y 52.551,Z 180,A 25.237,B 5.837,C 0.1714,E1 5.9863,E2 427.0403} C_DIS
LIN {X 121.2623,Y 55.5415,Z 180,A 26.6099,B 5.837,C 0.1682,E1 5.9847,E2 425.6706} C_DIS
LIN {X 119.8642,Y 58.4984,Z 180,A 27.9818,B 5.8372,C 0.1651,E1 5.9831,E2 424.302} C_DIS
LIN {X 118.3899,Y 61.4281,Z 180,A 29.343,B 5.8372,C 0.1623,E1 5.9813,E2 422.946} C_DIS
LIN {X 116.8438,Y 64.3222,Z 180,A 30.7406,B 5.8373,C 0.1589,E1 5.9795,E2 421.5492} C_DIS
LIN {X 115.2321,Y 67.1672,Z 180,A 32.1391,B 5.8374,C 0.1556,E1 5.9775,E2 420.1508} C_DIS
LIN {X 113.5509,Y 69.9713,Z 180,A 33.4996,B 5.8375,C 0.1528,E1 5.9756,E2 418.7951} C_DIS
LIN {X 111.7448,Y 72.8208,Z 180,A 34.9188,B 5.8375,C 0.1498,E1 5.9734,E2 417.379} C_DIS
LIN {X 109.9843,Y 75.453,Z 180,A 36.3842,B 5.8377,C 0.145,E1 5.9711,E2 415.9002} C_DIS
LIN {X 107.1991,Y 79.3611,Z 180,A 38.3946,B 5.8378,C 0.141,E1 5.9678,E2 413.8953} C_DIS
LIN {X 104.6093,Y 82.7452,Z 180,A 40.214,B 5.8379,C 0.137,E1 5.9647,E2 412.0767} C_DIS
LIN {X 102.0595,Y 85.8696,Z 180,A 41.8286,B 5.8379,C 0.135,E1 5.9618,E2 410.4758} C_DIS
LIN {X 99.375,Y 88.9624,Z 180,A 43.5,B 5.838,C 0.1325,E1 5.9588,E2 408.8145} C_DIS
LIN {X 96.6375,Y 91.9293,Z 180,A 45.203,B 5.838,C 0.1293,E1 5.9555,E2 407.1149} C_DIS
LIN {X 93.9547,Y 94.6691,Z 180,A 46.8625,B 5.8382,C 0.1258,E1 5.9523,E2 405.4535} C_DIS
LIN {X 91.3432,Y 97.1915,Z 180,A 48.4934,B 5.8382,C 0.1217,E1 5.9489,E2 403.8136} C_DIS
LIN {X 88.3256,Y 99.9415,Z 180,A 50.216,B 5.8382,C 0.1188,E1 5.9454,E2 402.0945} C_DIS
LIN {X 84.6563,Y 103.0685,Z 180,A 52.1164,B 5.8383,C 0.1174,E1 5.9413,E2 400.2144} C_DIS
LIN {X 81.4561,Y 105.6159,Z 180,A 53.7878,B 5.8383,C 0.1155,E1 5.9377,E2 398.5531} C_DIS
LIN {X 78.7767,Y 107.629,Z 180,A 55.4105,B 5.8385,C 0.1104,E1 5.934,E2 396.9082} C_DIS
LIN {X 75.452,Y 109.985,Z 180,A 56.9824,B 5.8385,C 0.1101,E1 5.9304,E2 395.3577} C_DIS
LIN {X 72.6459,Y 111.8583,Z 180,A 58.4107,B 5.8385,C 0.1081,E1 5.9271,E2 393.9317} C_DIS
LIN {X 69.9704,Y 113.5514,Z 180,A 59.7759,B 5.8385,C 0.1059,E1 5.9239,E2 392.566} C_DIS
LIN {X 67.0769,Y 115.2844,Z 180,A 61.1803,B 5.8385,C 0.1044,E1 5.9205,E2 391.1669} C_DIS
LIN {X 63.6051,Y 117.2356,Z 180,A 62.7295,B 5.8385,C 0.1042,E1 5.9168,E2 389.6371} C_DIS
LIN {X 61.3322,Y 118.4403,Z 180,A 64.1205,B 5.8387,C 0.0988,E1 5.9132,E2 388.2118} C_DIS
LIN {X 58.4032,Y 119.9111,Z 180,A 65.3654,B 5.8387,C 0.0993,E1 5.9102,E2 386.9866} C_DIS
LIN {X 55.4461,Y 121.3064,Z 180,A 66.7533,B 5.8387,C 0.0978,E1 5.9067,E2 385.6007} C_DIS
LIN {X 51.8448,Y 122.8883,Z 180,A 68.5798,B 5.8387,C 0.094,E1 5.9019,E2 383.7581} C_DIS
LIN {X 47.9102,Y 124.4749,Z 180,A 70.2285,B 5.8387,C 0.0944,E1 5.8977,E2 382.1304} C_DIS
LIN {X 44.9386,Y 125.5779,Z 180,A 71.5796,B 5.8387,C 0.0931,E1 5.8942,E2 380.7808} C_DIS
LIN {X 41.5926,Y 126.7265,Z 180,A 73.0731,B 5.8387,C 0.0921,E1 5.8902,E2 379.2907} C_DIS
LIN {X 38.6524,Y 127.6533,Z 180,A 74.3855,B 5.8387,C 0.0911,E1 5.8867,E2 377.9799} C_DIS
LIN {X 35.6499,Y 128.5239,Z 180,A 75.7307,B 5.8388,C 0.09,E1 5.8831,E2 376.6347} C_DIS
LIN {X 32.5311,Y 129.3485,Z 180,A 77.1937,B 5.8388,C 0.0879,E1 5.8791,E2 375.1629} C_DIS
LIN {X 29.2244,Y 130.1361,Z 180,A 78.5626,B 5.8388,C 0.0881,E1 5.8754,E2 373.8052} C_DIS
LIN {X 25.9156,Y 130.8362,Z 180,A 79.9964,B 5.8388,C 0.0875,E1 5.8715,E2 372.3742} C_DIS
LIN {X 22.8025,Y 131.4146,Z 180,A 81.3816,B 5.8388,C 0.0865,E1 5.8677,E2 370.9864} C_DIS
LIN {X 19.5728,Y 131.9344,Z 180,A 82.7722,B 5.8388,C 0.086,E1 5.8639,E2 369.598} C_DIS
LIN {X 16.3322,Y 132.3738,Z 180,A 84.1707,B 5.8388,C 0.0855,E1 5.86,E2 368.2007} C_DIS
LIN {X 13.0805,Y 132.734,Z 180,A 85.6099,B 5.8388,C 0.0846,E1 5.856,E2 366.758} C_DIS
LIN {X 9.708,Y 133.0228,Z 180,A 86.9913,B 5.8388,C 0.0852,E1 5.8522,E2 365.3857} C_DIS
LIN {X 5.7792,Y 133.2526,Z 180,A 88.8892,B 5.8389,C 0.0823,E1 5.8468,E2 363.4638} C_DIS
LIN {X 1.6465,Y 133.3677,Z 180,A 90.4835,B 5.8389,C 0.0844,E1 5.8424,E2 361.892} C_DIS
LIN {X -1.6411,Y 133.3677,Z 180,A 91.9319,B 5.8389,C 0.0839,E1 5.8383,E2 360.4399} C_DIS
Enddeposition()
END
